(* IEC 61131-3 sources: elnaProjects/ElpcLogic/PomarKc7Changed/build_USO_ecl (part 9) *)

  runDiProtection(protections.dPmaslo_gaz_less100);
  runDiProtection(protections.Reg_vozb_off);
  runDiProtection(protections.Fail_chastotnii_pusk);
  runDiProtection(protections.Off_avar_vikluchatel);
  runDiProtection(protections.AOKC_SHKC);
  runDiProtection(protections.AO_PRU);
  runDiProtection(protections.AO_ot_SHU);
  runDiProtection(protections.mvOff);
  runDiProtection(protections.Kran1_sdvig);
  runDiProtection(protections.Kran2_sdvig);
END_FUNCTION

FUNCTION anyProtectionInRemont : BOOL
  VAR_INPUT
    protections : ProtectionsConfig;
  END_VAR

  anyProtectioninRemont:=
  protections.Topornogo_podshipnika_EDT_1.Remont OR
  protections.Toy_podshipnika_EDT_2.Remont OR
  protections.Toy_podshipnika_kol_EDT_3.remont OR
  protections.Toy_podshipnika_kol_EDT_4.Remont OR
  protections.To_podshipnika_shest_red_EDT_5.Remont OR
  protections.To_podshipnika_shest_red_EDT_6.Remont OR
  protections.To_podshipnika_N_EDT_7.Remont OR
  protections.To_podshipnika_svob_konca_EDT_8.Remont OR
  protections.Ty_podshipnika_rab_kol_EDT_9.Remont OR
  protections.Typornogo_podshipnika_nerab_kolodok_HT_10.Remont OR
  protections.Tgaza_na_vyhode_H.Remont OR
  protections.Os_sdvig_nagnetatelja_plus.Remont OR
  protections.Os_sdvig_nagnetatelja_minus.Remont OR
  protections.Pgaza_na_vyhode_nagnetatelia_GPA_STOP.Remont OR
  protections.Pgaza_na_vhode_nagnetatelia_GPA_STOP.Remont OR
  protections.Pgaza_na_vyhode_nagnetatelia.Remont OR
  protections.dPmaslo_gaz.Remont OR
  protections.Pmaslo_sm_nizkoe.Remont OR
  protections.Pmaslo_sm_vysokoe.Remont OR
  protections.Vibro_skorost_OPED_T1.Remont OR
  protections.Vibro_skorost_OPED_T2.Remont OR
  protections.Vibro_skorost_OYP_kolesa_ED_T3.Remont OR
  protections.Vibro_skorost_OP_kolesa_RH_T4.Remont OR
  protections.Vibro_skorost_OP_shesterni_RED_T5.Remont OR
  protections.Vibro_skorost_OP_shesterni_RED_T6.Remont OR
  protections.dPmaslo_gaz_less100.Remont OR
  protections.Reg_vozb_off.Remont OR
  protections.Fail_chastotnii_pusk.Remont OR
  protections.Off_avar_vikluchatel.Remont OR
  protections.AOKC_SHKC.Remont OR
  protections.AO_PRU.Remont OR
  protections.AO_ot_SHU.Remont OR
  protections.mvOff.Remont OR
  protections.Kran1_sdvig.Remont OR
  protections.Kran2_sdvig.Remont;
END_FUNCTION

FUNCTION ResetAllSignaling : BOOL
  VAR_IN_OUT
    protections : ProtectionsConfig;
  END_VAR

  IF protections.Topornogo_podshipnika_EDT_1.Signaling THEN
      resetAiProtection(protections.Topornogo_podshipnika_EDT_1);  END_IF;

  IF protections.Toy_podshipnika_EDT_2.Signaling THEN
      resetAiProtection(protections.Toy_podshipnika_EDT_2); END_IF;

  IF protections.Toy_podshipnika_kol_EDT_3.Signaling THEN
      resetAiProtection(protections.Toy_podshipnika_kol_EDT_3); END_IF;

  IF protections.Toy_podshipnika_kol_EDT_4.Signaling THEN
      resetAiProtection(protections.Toy_podshipnika_kol_EDT_4); END_IF;

  IF protections.To_podshipnika_shest_red_EDT_5.Signaling THEN
      resetAiProtection(protections.To_podshipnika_shest_red_EDT_5); END_IF;

  IF protections.To_podshipnika_shest_red_EDT_6.Signaling THEN
      resetAiProtection(protections.To_podshipnika_shest_red_EDT_6); END_IF;

  IF protections.To_podshipnika_N_EDT_7.Signaling THEN
      resetAiProtection(protections.To_podshipnika_N_EDT_7); END_IF;

  IF protections.To_podshipnika_svob_konca_EDT_8.Signaling THEN
      resetAiProtection(protections.To_podshipnika_svob_konca_EDT_8); END_IF;

  IF protections.Ty_podshipnika_rab_kol_EDT_9.Signaling THEN
      resetAiProtection(protections.Ty_podshipnika_rab_kol_EDT_9); END_IF;

  IF protections.Typornogo_podshipnika_nerab_kolodok_HT_10.Signaling THEN
      resetAiProtection(protections.Typornogo_podshipnika_nerab_kolodok_HT_10); END_IF;

  IF protections.Tgaza_na_vyhode_H.Signaling THEN
      resetAiProtection(protections.Tgaza_na_vyhode_H); END_IF;

  IF protections.Os_sdvig_nagnetatelja_plus.Signaling THEN
     resetAiProtection(protections.Os_sdvig_nagnetatelja_plus); END_IF;

  IF protections.Os_sdvig_nagnetatelja_minus.Signaling THEN
      resetAiProtection(protections.Os_sdvig_nagnetatelja_minus); END_IF;

  IF protections.Pgaza_na_vyhode_nagnetatelia_GPA_STOP.Signaling THEN
      resetAiProtection(protections.Pgaza_na_vyhode_nagnetatelia_GPA_STOP); END_IF;

  IF protections.Pgaza_na_vhode_nagnetatelia_GPA_STOP.Signaling THEN
      resetAiProtection(protections.Pgaza_na_vhode_nagnetatelia_GPA_STOP); END_IF;

  IF protections.Pgaza_na_vyhode_nagnetatelia.Signaling THEN
      resetAiProtection(protections.Pgaza_na_vyhode_nagnetatelia); END_IF;

  IF protections.dPmaslo_gaz.Signaling THEN
      resetAiProtection(protections.dPmaslo_gaz); END_IF;

  IF protections.Pmaslo_sm_nizkoe.Signaling THEN
      resetAiProtection(protections.Pmaslo_sm_nizkoe); END_IF;

  IF protections.Pmaslo_sm_vysokoe.Signaling THEN
      resetAiProtection(protections.Pmaslo_sm_vysokoe); END_IF;

  IF protections.Vibro_skorost_OPED_T1.Signaling THEN
      resetAiProtection(protections.Vibro_skorost_OPED_T1); END_IF;

  IF protections.Vibro_skorost_OPED_T2.Signaling THEN
      resetAiProtection(protections.Vibro_skorost_OPED_T2); END_IF;

  IF protections.Vibro_skorost_OYP_kolesa_ED_T3.Signaling THEN
      resetAiProtection(protections.Vibro_skorost_OYP_kolesa_ED_T3); END_IF;

  IF protections.Vibro_skorost_OP_kolesa_RH_T4.Signaling THEN
      resetAiProtection(protections.Vibro_skorost_OP_kolesa_RH_T4); END_IF;

  IF protections.Vibro_skorost_OP_shesterni_RED_T5.Signaling THEN
      resetAiProtection(protections.Vibro_skorost_OP_shesterni_RED_T5); END_IF;

  IF protections.Vibro_skorost_OP_shesterni_RED_T6.Signaling THEN
      resetAiProtection(protections.Vibro_skorost_OP_shesterni_RED_T6); END_IF;

  IF protections.dPmaslo_gaz_less100.Signaling THEN
      resetDiProtection(protections.dPmaslo_gaz_less100); END_IF;

  IF protections.Reg_vozb_off.Signaling THEN
      resetDiProtection(protections.Reg_vozb_off); END_IF;

  IF protections.Fail_chastotnii_pusk.Signaling THEN
      resetDiProtection(protections.Fail_chastotnii_pusk); END_IF;

  IF protections.Off_avar_vikluchatel.Signaling THEN
      resetDiProtection(protections.Off_avar_vikluchatel); END_IF;

  IF protections.AOKC_SHKC.Signaling THEN
      resetDiProtection(protections.AOKC_SHKC); END_IF;

  IF protections.AO_PRU.Signaling THEN
      resetDiProtection(protections.AO_PRU); END_IF;

  IF protections.AO_ot_SHU.Signaling THEN
      resetDiProtection(protections.AO_ot_SHU); END_IF;

  IF protections.mvOff.Signaling THEN
      resetDiProtection(protections.mvOff); END_IF;

  IF protections.Kran1_sdvig.Signaling THEN
      resetDiProtection(protections.Kran1_sdvig); END_IF;

  IF protections.Kran2_sdvig.Signaling THEN
      resetDiProtection(protections.Kran2_sdvig); END_IF;
END_FUNCTION

FUNCTION_BLOCK fb_ProtectionsManager
  VAR
    cmd : BYTE;
  END_VAR
  VAR_IN_OUT
    str_PM : struct_ProtectionsManager;
  END_VAR
  VAR
    lastCmd : BYTE;
    autoRunPriznak : BOOL;
    onInit : BOOL;
  END_VAR
  VAR_EXTERNAL
    protections : ProtectionsConfig;
  END_VAR
  VAR
    timerUnBlock : TON;
    timerAutoRun : TON;
    UnBlockPriznak : BOOL;
  END_VAR

  IF NOT onInit THEN

      autoRunProtections(protections);
  onInit:=TRUE;
  END_IF;

  str_PM.protectionInRemont:=anyProtectioninRemont(protections);

  cmd := str_PM.inCommand;

  IF cmd <> 0 AND lastCmd <> cmd then
                UnBlockPriznak:=TRUE;
  	CASE BYTE_TO_INT(cmd) OF

  		(*RestartAllSignaling*) 1: 	ResetAllSignaling(protections);
  				          autoRunPriznak:=TRUE;

  	        (*RestartAllProtections*) 2: 	ResetAllProtections(protections);
                                                    autoRunPriznak:=TRUE;

                        (*CheckProtections*)  3: 	RunAllProtections(protections);

  	         (*ResetAllProtections*)  4: 	ResetAllProtections(protections);

  	END_CASE;

  END_IF;
  lastCmd := cmd;
  timerUnBlock(IN:=UnBlockPriznak, PT:=T#1S);
  timerAutoRun(IN:=autoRunPriznak, PT:=T#500MS);

  IF timerAutoRun.Q THEN autoRunProtections(protections);
  END_IF;

  IF timerUnBlock.Q THEN
  lastCmd:= 0;
  str_PM.inCommand:=0;
  autoRunPriznak:=FALSE;
  UnBlockPriznak:=FALSE;
  END_IF;
END_FUNCTION_BLOCK

FUNCTION stopPusk : BOOL
  VAR_IN_OUT
    algoritms : AlgoritmsConfig;
  END_VAR

  resetAndDisable(alg:=algoritms.Apusk);
  resetAndDisable(alg:=algoritms.SemiAutoPusk);
  resetAndDisable(alg:=algoritms.testPms);
  resetAndDisable(alg:=algoritms.puskV);
  resetAndDisable(alg:=algoritms.puskK);
  resetAndDisable(alg:=algoritms.testdPmg);
  resetAndDisable(alg:=algoritms.ppu);
  resetAndDisable(alg:=algoritms.puskOilSystem);
  resetAndDisable(alg:=algoritms.filling);
  resetAndDisable(alg:=algoritms.engineRun);
  resetAndDisable(alg:=algoritms.RingToLine);
  resetAndDisable(alg:=algoritms.LineToRing);
END_FUNCTION

FUNCTION anyDiscretPS : BOOL
  VAR_INPUT
    im : ImConfig;
  END_VAR

  anyDiscretPS:= TRUE;
      (*Im.SingleSignals.BEAO_srabotal.Q                     OR
      Im.SingleSignals.Vozb_ProboiVentila.Q	 OR
      Im.SingleSignals.Vozb_AsinchHod.Q	           OR
      Im.SingleSignals.NS_ForsingVozbugdenia.Q       OR
      Im.SingleSignals.Vozb_AutoUprVozbuditela_off.Q OR
      Im.SingleSignals.Vozb_KontaktorON.Q*)
END_FUNCTION

FUNCTION UnBlockAllProtections : BOOL
  VAR_IN_OUT
    protections : ProtectionsConfig;
  END_VAR

  protections.Topornogo_podshipnika_EDT_1.inOpcCommandsDisabled:=FALSE;
  protections.Toy_podshipnika_EDT_2.inOpcCommandsDisabled:=FALSE;
  protections.Toy_podshipnika_kol_EDT_3.inOpcCommandsDisabled:=FALSE;
  protections.Toy_podshipnika_kol_EDT_4.inOpcCommandsDisabled:=FALSE;
  protections.To_podshipnika_shest_red_EDT_5.inOpcCommandsDisabled:=FALSE;
  protections.To_podshipnika_shest_red_EDT_6.inOpcCommandsDisabled:=FALSE;
  protections.To_podshipnika_N_EDT_7.inOpcCommandsDisabled:=FALSE;
  protections.To_podshipnika_svob_konca_EDT_8.inOpcCommandsDisabled:=FALSE;
  protections.Ty_podshipnika_rab_kol_EDT_9.inOpcCommandsDisabled:=FALSE;
  protections.Typornogo_podshipnika_nerab_kolodok_HT_10.inOpcCommandsDisabled:=FALSE;
  protections.Tgaza_na_vyhode_H.inOpcCommandsDisabled:=FALSE;
  protections.Os_sdvig_nagnetatelja_plus.inOpcCommandsDisabled:=FALSE;
  protections.Os_sdvig_nagnetatelja_minus.inOpcCommandsDisabled:=FALSE;
  protections.Pgaza_na_vyhode_nagnetatelia_GPA_STOP.inOpcCommandsDisabled:=FALSE;
  protections.Pgaza_na_vhode_nagnetatelia_GPA_STOP.inOpcCommandsDisabled:=FALSE;
  protections.Pgaza_na_vyhode_nagnetatelia.inOpcCommandsDisabled:=FALSE;
  protections.dPmaslo_gaz.inOpcCommandsDisabled:=FALSE;
  protections.Pmaslo_sm_nizkoe.inOpcCommandsDisabled:=FALSE;
  protections.Pmaslo_sm_vysokoe.inOpcCommandsDisabled:=FALSE;
  protections.Vibro_skorost_OPED_T1.inOpcCommandsDisabled:=FALSE;
  protections.Vibro_skorost_OPED_T2.inOpcCommandsDisabled:=FALSE;
  protections.Vibro_skorost_OYP_kolesa_ED_T3.inOpcCommandsDisabled:=FALSE;
  protections.Vibro_skorost_OP_kolesa_RH_T4.inOpcCommandsDisabled:=FALSE;
  protections.Vibro_skorost_OP_shesterni_RED_T5.inOpcCommandsDisabled:=FALSE;
  protections.Vibro_skorost_OP_shesterni_RED_T6.inOpcCommandsDisabled:=FALSE;
  protections.dPmaslo_gaz_less100.inOpcCommandsDisabled:=FALSE;
  protections.Reg_vozb_off.inOpcCommandsDisabled:=FALSE;
  protections.Fail_chastotnii_pusk.inOpcCommandsDisabled:=FALSE;
  protections.Off_avar_vikluchatel.inOpcCommandsDisabled:=FALSE;
  protections.AOKC_SHKC.inOpcCommandsDisabled:=FALSE;
  protections.AO_PRU.inOpcCommandsDisabled:=FALSE;
  protections.AO_ot_SHU.inOpcCommandsDisabled:=FALSE;
  protections.mvOff.inOpcCommandsDisabled:=FALSE;
  protections.Kran1_sdvig.inOpcCommandsDisabled:=FALSE;
  protections.Kran2_sdvig.inOpcCommandsDisabled:=FALSE;
END_FUNCTION

FUNCTION_BLOCK fb_AlgoritmsManager
  VAR_IN_OUT
    str_AM : struct_AlgoritmsManager;
  END_VAR
  VAR
    onInit : BOOL;
  END_VAR
  VAR_EXTERNAL
    ai : AiConfig;
  END_VAR
  VAR
    EoTrig : R_TRIG;
    EoFTrig : F_TRIG;
    PsLampTrig : R_TRIG;
    PsLampFTrig : F_TRIG;
    Ring : R_TRIG;
    Line : R_TRIG;
    statusDualInput : TYPE_statusDualInput;
  END_VAR
  VAR_EXTERNAL
    IM : ImConfig;
    protections : ProtectionsConfig;
    algoritms : AlgoritmsConfig;
    ModeGpa : TYPE_ModeGpa;
  END_VAR

  IF NOT onInit THEN
            DisableAiLimits(ai);
            (*IM.SingleSignals.P_oil_low.Disabled_Sig:=TRUE;
            IM.SingleSignals.dP_oilgaz_low.Disabled_Sig:=TRUE;*)
            str_AM.nMode:=ModeGpa.MODE_STOP;
            BlockAllIM(IM);
            runIfNotRunning(algoritms.AutoTen);
  onInit:=TRUE;
  END_IF;

  str_AM.DiscretPS:=anyDiscretPS(IM);
  str_AM.AnalogsPs:=anyAnalogsPs(ai);
  str_AM.ProtectionSignaling:=anyProtectionSignaling(protections);

  (*EoTrig(CLK := IM.SingleSignals.BEO_Srabat.Q);*)
  IF EoTrig.Q THEN
  	stopPusk(algoritms);
  	resetAndDisable(algoritms.Remont);
  	resetAndDisable(algoritms.no);
  	resetAndDisable(algoritms.ao);
  	str_AM.nMode:=ModeGpa.MODE_EO;
  END_IF;
  (*EoFTrig(CLK := IM.SingleSignals.BEO_Srabat.Q);*)
  IF EoFTrig.Q THEN
  	str_AM.nMode:=ModeGpa.MODE_STOP;
  	runIfNotRunning(algoritms.ao);
  END_IF;

  (*IF (str_AM.ProtectionSignaling OR Im.SingleSignals.AO_KC.Q OR Im.SingleSignals.AOGPA_knopkaSHU.Q OR Im.SingleSignals.AOGPA_PRU.Q )
  	AND NOT((str_AM.mode=ModeGpa.MODE_AO) OR (str_AM.mode=ModeGpa.MODE_EO) OR IM.SingleOutputs.IndikicijaAS_fonar.Q
            OR (str_AM.mode=ModeGpa.MODE_TESTAZ) OR (str_AM.mode=ModeGpa.MODE_TESTDPMG) OR (str_AM.mode=ModeGpa.MODE_REMONT) OR
            (str_AM.mode=ModeGpa.MODE_TESTPMS))THEN
  		runIfNotRunning(algoritms.ao);
  	str_AM.nMode:=ModeGpa.MODE_AO;
  END_IF;
  *)
  (*IF Im.SingleSignals.NOGPA_knopkaSHU.Q  AND algoritms.no.CanRun THEN
  	runIfNotRunning(algoritms.no);
            str_AM.nMode:=ModeGpa.MODE_NO;
  END_IF;*)

  PsLampTrig(CLK := str_AM.DiscretPS OR str_AM.AnalogsPs);
  (*IF PsLampTrig.Q THEN
            runIfNotRunningSO(IM.SingleOutputs.IndikicijaPS_fonar);
  END_IF;*)
  PsLampFTrig(CLK := str_AM.DiscretPS OR str_AM.AnalogsPs);
  (*IF PsLampFTrig.Q THEN
            resetIfRunningSO(IM.SingleOutputs.IndikicijaPS_fonar);
  END_IF;*)

  IF str_AM.mode = ModeGpa.MODE_WORK_Line OR str_AM.mode = ModeGpa.MODE_WORK_Ring  THEN

  	Ring(CLK:=Im.kran6.onStatus=statusDualInput.STATUS_On);
  	Line(CLK:=Im.kran6.onStatus=statusDualInput.STATUS_Off);

  	IF Ring.Q AND str_AM.mode = ModeGpa.MODE_WORK_Line THEN
  		str_AM.nMode:=ModeGpa.MODE_WORK_Ring;
  	END_IF;
  	IF Line.Q AND str_AM.mode = ModeGpa.MODE_WORK_Ring THEN
  		str_AM.nMode:=ModeGpa.MODE_WORK_Line;
  	END_IF;

  END_IF;

  IF str_AM.mode = ModeGpa.MODE_WORK_Line THEN
            runIfNotRunning(alg:=algoritms.AntiPompag);
  	ELSE
            resetAndDisable(alg:=algoritms.AntiPompag);
  END_IF;

  IF str_AM.nMode<>str_AM.mode THEN
  	str_AM.mode:=str_AM.nMode;
  	CASE str_AM.mode OF
  	(*ModeGpa.MODE_REMONT*)1:
  		stopPusk(algoritms);
  		resetAndDisable(alg:=algoritms.no);
  		resetAndDisable(alg:=algoritms.ao);
  		resetAndDisable(alg:=algoritms.TestProtection);
                      resetAndDisable(alg:=algoritms.testIm);

  	(*ModeGpa.MODE_TESTAZ*)16:
  		stopPusk(algoritms);
  		resetAndDisable(alg:=algoritms.ao);
  		resetAndDisable(alg:=algoritms.no);
                      resetAndDisable(alg:=algoritms.Remont);
                      resetAndDisable(alg:=algoritms.testIm);

            (*ModeGpa.MODE_TESTIM*)15:
                      stopPusk(algoritms);
                      resetAndDisable(alg:=algoritms.Remont);
                      resetAndDisable(alg:=algoritms.TestProtection);

  	(*ModeGpa.MODE_EO*)14:
  		stopPusk(algoritms);
  		resetAndDisable(alg:=algoritms.no);
  		resetAndDisable(alg:=algoritms.ao);
  		resetAndDisable(alg:=algoritms.Remont);
                      resetAndDisable(alg:=algoritms.testIm);
                      resetAndDisable(alg:=algoritms.TestProtection);
  	(*ModeGpa.MODE_AO*)13:
  		(*//stopPusk();*)
  		resetAndDisable(alg:=algoritms.no);
  		resetAndDisable(alg:=algoritms.Remont);
                      resetAndDisable(alg:=algoritms.testIm);
                      resetAndDisable(alg:=algoritms.TestProtection);
                      algoritms.VibegPNS.inCanRun:=TRUE;
  	(*ModeGpa.MODE_NO*)12:
  		stopPusk(algoritms);
                      resetAndDisable(alg:=algoritms.testIm);
                      resetAndDisable(alg:=algoritms.Remont);
                      resetAndDisable(alg:=algoritms.TestProtection);
                      algoritms.VibegPNS.inCanRun:=TRUE;
  		algoritms.ao.inCanRun:=TRUE;
  	(*ModeGpa.MODE_APUSK*)8:
  		resetAndDisable(alg:=algoritms.SemiAutoPusk);
  		resetAndDisable(alg:=algoritms.puskV);
  		resetAndDisable(alg:=algoritms.puskK);
  		resetAndDisable(alg:=algoritms.testdPmg);
  		resetAndDisable(alg:=algoritms.testPms);
  		(*resetAndDisable(alg:=algoritms.testIm);
                      resetAndDisable(alg:=algoritms.TestProtection);
                      resetAndDisable(alg:=algoritms.Remont);*)
  		resetAndDisable(alg:=algoritms.ppu);
  		algoritms.no.inCanRun:=TRUE;
  		algoritms.ao.inCanRun:=TRUE;

  	(*ModeGpa.MODE_MPUSK*)9:
  		resetAndDisable(alg:=algoritms.Apusk);
  		resetAndDisable(alg:=algoritms.puskV);
  		resetAndDisable(alg:=algoritms.puskK);
  		resetAndDisable(alg:=algoritms.testdPmg);
  		resetAndDisable(alg:=algoritms.testPms);
  		(*resetAndDisable(alg:=algoritms.testIm);
                      resetAndDisable(alg:=algoritms.TestProtection);
                      resetAndDisable(alg:=algoritms.Remont);	*)
  		resetAndDisable(alg:=algoritms.ppu);
  		algoritms.no.inCanRun:=TRUE;
                      algoritms.no.inOpcCommandsDisabled:=FALSE;
  		algoritms.ao.inCanRun:=TRUE;
                      algoritms.ao.inOpcCommandsDisabled:=FALSE;

  	(*ModeGpa.MODE_PUSKK*)5:
                      resetAndDisable(alg:=algoritms.ppu);
  		resetAndDisable(alg:=algoritms.Apusk);
  		resetAndDisable(alg:=algoritms.SemiAutoPusk);
  		resetAndDisable(alg:=algoritms.TestProtection);
                      resetAndDisable(alg:=algoritms.Remont);
  		resetAndDisable(alg:=algoritms.testIm	 );
  		algoritms.no.inCanRun:=TRUE;
                      algoritms.no.inOpcCommandsDisabled:=FALSE;
  		algoritms.ao.inCanRun:=TRUE;
                      algoritms.ao.inOpcCommandsDisabled:=FALSE;
  	(*ModeGpa.MODE_PUSKV*)4:
                      resetAndDisable(alg:=algoritms.ppu);
  		resetAndDisable(alg:=algoritms.Apusk);
  		resetAndDisable(alg:=algoritms.SemiAutoPusk);
  		resetAndDisable(alg:=algoritms.TestProtection);
                      resetAndDisable(alg:=algoritms.Remont);
  		resetAndDisable(alg:=algoritms.testIm	 );
  		algoritms.no.inCanRun:=TRUE;
                      algoritms.no.inOpcCommandsDisabled:=FALSE;
  		algoritms.ao.inCanRun:=TRUE;
                      algoritms.ao.inOpcCommandsDisabled:=FALSE;

  	(*ModeGpa.MODE_TESTDPMG*)6:
                      resetAndDisable(alg:=algoritms.ppu);
  		resetAndDisable(alg:=algoritms.Apusk);
  		resetAndDisable(alg:=algoritms.SemiAutoPusk);
  		resetAndDisable(alg:=algoritms.TestProtection);
                      resetAndDisable(alg:=algoritms.Remont);
  		resetAndDisable(alg:=algoritms.testIm	 );
  		algoritms.no.inCanRun:=TRUE;
                      algoritms.no.inOpcCommandsDisabled:=FALSE;
  		algoritms.ao.inCanRun:=TRUE;
                      algoritms.ao.inOpcCommandsDisabled:=FALSE;

  	(*ModeGpa.MODE_TESTPMS*)7:
                      resetAndDisable(alg:=algoritms.ppu);
  		resetAndDisable(alg:=algoritms.Apusk);
  		resetAndDisable(alg:=algoritms.SemiAutoPusk);
  		resetAndDisable(alg:=algoritms.TestProtection);
                      resetAndDisable(alg:=algoritms.Remont);
  		resetAndDisable(alg:=algoritms.testIm);
  		algoritms.no.inCanRun:=TRUE;
                      algoritms.no.inOpcCommandsDisabled:=FALSE;
  		algoritms.ao.inCanRun:=TRUE;
                      algoritms.ao.inOpcCommandsDisabled:=FALSE;

  	(*ModeGpa.MODE_WORK_Ring*)10:
  		resetAndDisable(alg:=algoritms.Apusk);
  		resetAndDisable(alg:=algoritms.SemiAutoPusk);
  		resetAndDisable(alg:=algoritms.puskV);
  		resetAndDisable(alg:=algoritms.puskK);
  		resetAndDisable(alg:=algoritms.testdPmg);
  		resetAndDisable(alg:=algoritms.testPms);
  		resetAndDisable(alg:=algoritms.ppu);
  		algoritms.no.inCanRun:=TRUE;
                      algoritms.no.inOpcCommandsDisabled:=FALSE;
  		algoritms.ao.inCanRun:=TRUE;
                      algoritms.ao.inOpcCommandsDisabled:=FALSE;

  	(*ModeGpa.MODE_WORK_Line*)11:
  		resetAndDisable(alg:=algoritms.Apusk);
  		resetAndDisable(alg:=algoritms.SemiAutoPusk);
  		resetAndDisable(alg:=algoritms.puskV);
  		resetAndDisable(alg:=algoritms.puskK);
  		resetAndDisable(alg:=algoritms.testdPmg);
  		resetAndDisable(alg:=algoritms.testPms);
  		resetAndDisable(alg:=algoritms.ppu);
  		resetAndDisable(alg:=algoritms.testIm	 );
  		algoritms.no.inCanRun:=TRUE;
                      algoritms.no.inOpcCommandsDisabled:=FALSE;
  		algoritms.ao.inCanRun:=TRUE;
                      algoritms.ao.inOpcCommandsDisabled:=FALSE;

  	(*ModeGpa.MODE_STOP*)2:
  		algoritms.ppu.inCanRun:=TRUE;
                      runIfNotRunning(alg:=algoritms.ppu);
  		algoritms.no.inCanRun:=TRUE;
                      algoritms.no.inOpcCommandsDisabled:=FALSE;
  		algoritms.ao.inCanRun:=TRUE;
                      algoritms.ao.inOpcCommandsDisabled:=FALSE;
                      (*UnBlockAllProtections(protections);*)
  		BlockAllIM(IM);
  		algoritms.Remont.inCanRun:=TRUE;
  		algoritms.Remont.inOpcCommandsDisabled:=FALSE;
  		algoritms.testim.inCanRun:=TRUE;
  		algoritms.testim.inOpcCommandsDisabled:=FALSE;
  		algoritms.TestProtection.inCanRun:=TRUE;
  		algoritms.TestProtection.inOpcCommandsDisabled:=FALSE;
                      algoritms.VibegPNS.inCanRun:=FALSE;
                      algoritms.AutoAvom.inCanRun:=FALSE;
  		(*resetAndDisable(alg:=algoritms.puskV);
  		resetAndDisable(alg:=algoritms.puskK);
  		resetAndDisable(alg:=algoritms.testdPmg);
  		resetAndDisable(alg:=algoritms.testPms);*)
  	(*ModeGpa.MODE_READY*)3:
  		resetAndDisable(alg:=algoritms.Remont);
  		resetAndDisable(alg:=algoritms.testim);
  		resetAndDisable(alg:=algoritms.TestProtection);
                      algoritms.Apusk.inCanRun:=TRUE;
                      algoritms.Apusk.inOpcCommandsDisabled:=FALSE;
  		algoritms.SemiAutoPusk.inCanRun:=TRUE;
                      algoritms.SemiAutoPusk.inOpcCommandsDisabled:=FALSE;
  	END_CASE;
  END_IF;
END_FUNCTION_BLOCK

FUNCTION remontAllProtections : BOOL
  VAR_IN_OUT
    protections : ProtectionsConfig;
  END_VAR
  VAR CONSTANT
    cmdRemont : WORD          := 4;
  END_VAR

  protections.Topornogo_podshipnika_EDT_1.inCommand_Alg:=cmdRemont;
  protections.Toy_podshipnika_EDT_2.inCommand_Alg:=cmdRemont;
  protections.Toy_podshipnika_kol_EDT_3.inCommand_Alg:=cmdRemont;
  protections.Toy_podshipnika_kol_EDT_4.inCommand_Alg:=cmdRemont;
  protections.To_podshipnika_shest_red_EDT_5.inCommand_Alg:=cmdRemont;
  protections.To_podshipnika_shest_red_EDT_6.inCommand_Alg:=cmdRemont;
  protections.To_podshipnika_N_EDT_7.inCommand_Alg:=cmdRemont;
  protections.To_podshipnika_svob_konca_EDT_8.inCommand_Alg:=cmdRemont;
  protections.Ty_podshipnika_rab_kol_EDT_9.inCommand_Alg:=cmdRemont;
  protections.Typornogo_podshipnika_nerab_kolodok_HT_10.inCommand_Alg:=cmdRemont;
  protections.Tgaza_na_vyhode_H.inCommand_Alg:=cmdRemont;
  protections.Os_sdvig_nagnetatelja_plus.inCommand_Alg:=cmdRemont;
  protections.Os_sdvig_nagnetatelja_minus.inCommand_Alg:=cmdRemont;
  protections.Pgaza_na_vyhode_nagnetatelia_GPA_STOP.inCommand_Alg:=cmdRemont;
  protections.Pgaza_na_vhode_nagnetatelia_GPA_STOP.inCommand_Alg:=cmdRemont;
  protections.Pgaza_na_vyhode_nagnetatelia.inCommand_Alg:=cmdRemont;
  protections.dPmaslo_gaz.inCommand_Alg:=cmdRemont;
  protections.Pmaslo_sm_nizkoe.inCommand_Alg:=cmdRemont;
  protections.Pmaslo_sm_vysokoe.inCommand_Alg:=cmdRemont;
  protections.Vibro_skorost_OPED_T1.inCommand_Alg:=cmdRemont;
  protections.Vibro_skorost_OPED_T2.inCommand_Alg:=cmdRemont;
  protections.Vibro_skorost_OYP_kolesa_ED_T3.inCommand_Alg:=cmdRemont;
  protections.Vibro_skorost_OP_kolesa_RH_T4.inCommand_Alg:=cmdRemont;
  protections.Vibro_skorost_OP_shesterni_RED_T5.inCommand_Alg:=cmdRemont;
  protections.Vibro_skorost_OP_shesterni_RED_T6.inCommand_Alg:=cmdRemont;
  protections.dPmaslo_gaz_less100.inCommand_Alg:=cmdRemont;
  protections.Reg_vozb_off.inCommand_Alg:=cmdRemont;
  protections.Fail_chastotnii_pusk.inCommand_Alg:=cmdRemont;
  protections.Off_avar_vikluchatel.inCommand_Alg:=cmdRemont;
  protections.AOKC_SHKC.inCommand_Alg:=cmdRemont;
  protections.AO_PRU.inCommand_Alg:=cmdRemont;
  protections.AO_ot_SHU.inCommand_Alg:=cmdRemont;
  protections.mvOff.inCommand_Alg:=cmdRemont;
  protections.Kran1_sdvig.inCommand_Alg:=cmdRemont;
  protections.Kran2_sdvig.inCommand_Alg:=cmdRemont;
END_FUNCTION

FUNCTION nsCepeiControl : BOOL
  VAR_INPUT
    im : ImConfig;
  END_VAR

  nsCepeiControl:= NOT (
  	im.kran1.reliability OR
  	im.kran2.reliability OR
  	im.kran4.reliability OR
  	im.kran5.reliability OR
  	im.kran6.reliability OR
  	im.kran3b.reliability OR
  	im.pns.reliability OR
  	im.nu1.reliability OR
  	im.nu2.reliability OR
  	im.PNS.reliability OR
            im.v1_Avom.reliability OR
            im.v2_Avom.reliability OR
            (*im.Ten.reliability OR*)
  	im.mv.reliability);
END_FUNCTION

FUNCTION NapryageniaOK : BOOL
  VAR_INPUT
    im : ImConfig;
  END_VAR

  NapryageniaOK:=
  NOT (Im.SingleSignals.NS_G1_G2.Q
  OR Im.SingleSignals.NS_G10_G11.Q
  OR Im.SingleSignals.NS_G13_G14.Q
  OR Im.SingleSignals.NS_G15_G16.Q
  OR Im.SingleSignals.NS_G17.Q
  OR Im.SingleSignals.NS_G18_G19.Q
  OR Im.SingleSignals.NS_G3_G4.Q
  OR Im.SingleSignals.NS_G5_G6.Q
  OR Im.SingleSignals.NS_G7_G8.Q
  OR im.SingleSignals.QF1_on.Q
  OR Im.SingleSignals.QF2_on.Q
  OR Im.SingleSignals.QF23_on.Q
  OR Im.SingleSignals.QF4_QF5_on.Q
  OR Im.SingleSignals.QF6_QF7_on.Q
  OR Im.SingleSignals.QF8_QF9_on.Q
  OR Im.SingleSignals.QF10_QF11_on.Q
  OR im.SingleSignals.QF12_QF13_on.Q
  OR im.SingleSignals.QF22_on.Q
  OR Im.SingleSignals.QF14_QF15_on.Q);
END_FUNCTION

FUNCTION discretNS : BOOL
  VAR_INPUT
    di : DiConfig;
  END_VAR

  discretNS:=  ((di.di_0.reliability <> 255)
                OR (di.di_1.reliability <> 255)
                OR (di.di_2.reliability <> 255)
                OR (di.di_3.reliability <> 255)
                OR (di.di_4.reliability <> 255)
                OR (di.di_5.reliability <> 255)
                OR (di.di_6.reliability <> 255)
                OR (di.di_7.reliability <> 255)
                OR (di.di_8.reliability <> 255)
                OR (di.di_9.reliability <> 255)
                OR (di.di_10.reliability <> 255)
                OR (di.di_11.reliability <> 255)
                OR (di.di_12.reliability <> 255)
                OR (di.di_13.reliability <> 255)
                OR (di.di_14.reliability <> 255));
               (* OR (di.di_15.reliability <> 255)); *)
END_FUNCTION

FUNCTION BlockAllProtections : BOOL
  VAR_IN_OUT
    protections : ProtectionsConfig;
  END_VAR

  protections.Topornogo_podshipnika_EDT_1.inOpcCommandsDisabled:=TRUE;
  protections.Toy_podshipnika_EDT_2.inOpcCommandsDisabled:=TRUE;
  protections.Toy_podshipnika_kol_EDT_3.inOpcCommandsDisabled:=TRUE;
  protections.Toy_podshipnika_kol_EDT_4.inOpcCommandsDisabled:=TRUE;
  protections.To_podshipnika_shest_red_EDT_5.inOpcCommandsDisabled:=TRUE;
  protections.To_podshipnika_shest_red_EDT_6.inOpcCommandsDisabled:=TRUE;
  protections.To_podshipnika_N_EDT_7.inOpcCommandsDisabled:=TRUE;
  protections.To_podshipnika_svob_konca_EDT_8.inOpcCommandsDisabled:=TRUE;
  protections.Ty_podshipnika_rab_kol_EDT_9.inOpcCommandsDisabled:=TRUE;
  protections.Typornogo_podshipnika_nerab_kolodok_HT_10.inOpcCommandsDisabled:=TRUE;
  protections.Tgaza_na_vyhode_H.inOpcCommandsDisabled:=TRUE;
  protections.Os_sdvig_nagnetatelja_plus.inOpcCommandsDisabled:=TRUE;
  protections.Os_sdvig_nagnetatelja_minus.inOpcCommandsDisabled:=TRUE;
  protections.Pgaza_na_vyhode_nagnetatelia_GPA_STOP.inOpcCommandsDisabled:=TRUE;
  protections.Pgaza_na_vhode_nagnetatelia_GPA_STOP.inOpcCommandsDisabled:=TRUE;
  protections.Pgaza_na_vyhode_nagnetatelia.inOpcCommandsDisabled:=TRUE;
  protections.dPmaslo_gaz.inOpcCommandsDisabled:=TRUE;
  protections.Pmaslo_sm_nizkoe.inOpcCommandsDisabled:=TRUE;
  protections.Pmaslo_sm_vysokoe.inOpcCommandsDisabled:=TRUE;
  protections.Vibro_skorost_OPED_T1.inOpcCommandsDisabled:=TRUE;
  protections.Vibro_skorost_OPED_T2.inOpcCommandsDisabled:=TRUE;
  protections.Vibro_skorost_OYP_kolesa_ED_T3.inOpcCommandsDisabled:=TRUE;
  protections.Vibro_skorost_OP_kolesa_RH_T4.inOpcCommandsDisabled:=TRUE;
  protections.Vibro_skorost_OP_shesterni_RED_T5.inOpcCommandsDisabled:=TRUE;
  protections.Vibro_skorost_OP_shesterni_RED_T6.inOpcCommandsDisabled:=TRUE;
  protections.dPmaslo_gaz_less100.inOpcCommandsDisabled:=TRUE;
  protections.Reg_vozb_off.inOpcCommandsDisabled:=TRUE;
  protections.Fail_chastotnii_pusk.inOpcCommandsDisabled:=TRUE;
  protections.Off_avar_vikluchatel.inOpcCommandsDisabled:=TRUE;
  protections.AOKC_SHKC.inOpcCommandsDisabled:=TRUE;
  protections.AO_PRU.inOpcCommandsDisabled:=TRUE;
  protections.AO_ot_SHU.inOpcCommandsDisabled:=TRUE;
  protections.mvOff.inOpcCommandsDisabled:=TRUE;
  protections.Kran1_sdvig.inOpcCommandsDisabled:=TRUE;
  protections.Kran2_sdvig.inOpcCommandsDisabled:=TRUE;
END_FUNCTION

PROGRAM program0
  VAR
    SysTime : LREAL;
    systime_ns : ULINT;
    systime_s : ULINT;
    preSysTime : LREAL;
    tmpCycle : LREAL;
    preSys_s : ULINT;
    preSys_ns : ULINT;
  END_VAR
  VAR_EXTERNAL
    cur_Cycle : REAL;
    gStart_Tmr : REAL;
  END_VAR
  VAR
    Timings : fb_Timings;
    _init : BOOL          := TRUE;
    life_count : UINT;
    AI_structs_ini : proc_AI_Init;
    AI_Proc : proc_AI;
    AO_structs_ini : proc_AO_Init;
    AO_Proc : proc_AO;
    DI_structs_ini : proc_DI_Init;
    DI_Proc : proc_DI;
    DO_structs_ini : proc_DO_Init;
    DO_Proc : proc_DO;
    Get_algoritms_OPC : OPC_algoritms_set;
    Set_algoritms_OPC : OPC_algoritms_get;
    IM_structs_ini : proc_IM_Init;
    IM_Proc : proc_IM;
    Protections_structs_ini : proc_Protections_Init;
    Protections_Proc : proc_Protection;
    Algoritms_Proc : proc_algoritms;
    AlgoritmsManager : fb_AlgoritmsManager;
    ProtectionsManager : fb_ProtectionsManager;
  END_VAR
  VAR_EXTERNAL
    algManager : struct_AlgoritmsManager;
    protectManager : struct_ProtectionsManager;
  END_VAR

  (* Обработка времени. *)
  SysTime := ULINT_TO_LREAL(systime_s) + (1.0E-9 * ULINT_TO_LREAL(systime_ns));
  preSysTime := SysTime;
  tmpCycle := ULINT_TO_LREAL(systime_s - preSys_s) + 1.0E-9 * (ULINT_TO_LREAL(systime_ns) - ULINT_TO_LREAL(preSys_ns));
  cur_Cycle := LREAL_TO_REAL(tmpCycle);
  preSys_s := systime_s;
  preSys_ns := systime_ns;
  IF gStart_Tmr < 99999.9 THEN gStart_Tmr := gStart_Tmr + cur_Cycle; END_IF;
  Timings();

  IF  _init (*or external_init_ai *) then           (* Требуется инициализация структур и ФБ. *)
    (* Инициализация аналоговых входов. *)
      AI_structs_ini(init := TRUE);
      AI_Proc((*init := FALSE*));

    (* Инициализация дискретных входов. *)
      DI_structs_ini(init := TRUE);
      DI_Proc((*init := FALSE*));

      (* Инициализация аналоговых выходов. *)
  (*     AO_structs_ini(init := TRUE);
         AO_Proc(init := TRUE);*)

    (* Инициализация дискретных выходов. *)
      DO_structs_ini(init := TRUE);
      DO_Proc((*init := FALSE*));

     (* Инициализация ИМ. *)
      IM_structs_ini(init := TRUE);
      IM_Proc();

     (* Инициализация Защит *)
      Protections_structs_ini(init := TRUE);
      (*Protections_Proc();*)

       (* Стартовая инициализация OPC-тэгов элементами канальных структур. *)
          (*___________________AI______________________________________________________________________________*)
      (*ini_AI_OPC();*)

      _init := FALSE;

    ELSE                         (* Завершена инициализация структур и ФБ. *)

  (* Перенос OPC-тэгов в элементы структур каналов. *)
        (*___________________________________________AI________________________________________________*)
      (*Get_AI_OPC(); *)
       Get_algoritms_OPC();

     (* Пересчёт защит САУ. *)
     ProtectionsManager(protectManager);

       (* Пересчёт алгоритмов САУ. *)
     AlgoritmsManager(algManager);

      (****               Опрос входов.              ****)
          (* Опрос аналоговых входов. *)
      AI_Proc((*init := FALSE*));

          (* Опрос дискретных входов. *)
      DI_Proc((*init := FALSE*));

      (****              Запись выходов.             ****)
          (* Запись аналоговых выходов. *)
  (*    AO_Proc(init := FALSE);*)

       (* Запись дискретных выходов. *)
      DO_Proc((*init := FALSE*));

      (****               Опрос ИМ              ****)
      IM_Proc();

      (****            Опрос Защит              ****)
      Protections_Proc();

      Algoritms_Proc();

  END_IF;

  (* Передача информации на верхний уровень по OPC UA протоколу. *)
    (* Передача состояний каналов AI. *)
  (*Set_AI_OPC();)*
  (* Передача состояний каналов ИМ. *)
  (* Передача состояний защит. *)
  (* Передача состояний алгоритмов. *)
  Set_algoritms_OPC();
END_PROGRAM

CONFIGURATION config1
  VAR_GLOBAL
    systime_s AT %IL0.10.10 : ULINT;
    systime_ns AT %IL0.10.11 : ULINT;
    current_retrieve_us AT %IL0.10.12 : ULINT;
    current_config_us AT %IL0.10.13 : ULINT;
    current_publish_us AT %IL0.10.14 : ULINT;
    current_run_us AT %IL0.10.15 : ULINT;
    max_retrieve_us AT %QL0.10.16 : ULINT;
    max_config_us AT %QL0.10.17 : ULINT;
    max_publish_us AT %QL0.10.18 : ULINT;
    plc_run_number AT %IL0.10.19 : ULINT;
    arAIN_0 : TItemAIN;
    arAIN_1 : TItemAIN;
    arAIN_2 : TItemAIN;
    arAIN_3 : TItemAIN;
    arAIN_4 : TItemAIN;
    arAIN_5 : TItemAIN;
    arAIN_6 : TItemAIN;
    arAIN_7 : TItemAIN;
    arAIN_8 : TItemAIN;
    arAIN_9 : TItemAIN;
    arAIN_10 : TItemAIN;
    arAIN_11 : TItemAIN;
    arAIN_12 : TItemAIN;
    arAIN_13 : TItemAIN;
    arAIN_14 : TItemAIN;
    arAIN_15 : TItemAIN;
    arAIN_16 : TItemAIN;
    arAIN_17 : TItemAIN;
    arAIN_18 : TItemAIN;
    arAIN_19 : TItemAIN;
    arAIN_20 : TItemAIN;
    arAIN_21 : TItemAIN;
    arAIN_22 : TItemAIN;
    arAIN_23 : TItemAIN;
    arAIN_24 : TItemAIN;
    arAIN_25 : TItemAIN;
    arAIN_26 : TItemAIN;
    arAIN_27 : TItemAIN;
    arAIN_28 : TItemAIN;
    arAIN_29 : TItemAIN;
    arAIN_30 : TItemAIN;
    arAIN_31 : TItemAIN;
    arAIN_32 : TItemAIN;
    arAIN_33 : TItemAIN;
    arAIN_34 : TItemAIN;
    arAIN_35 : TItemAIN;
    arAIN_36 : TItemAIN;
    arAIN_37 : TItemAIN;
    arAIN_38 : TItemAIN;
    arAIN_39 : TItemAIN;
    arAIN_40 : TItemAIN;
    arAIN_41 : TItemAIN;
    arAIN_42 : TItemAIN;
    arAIN_43 : TItemAIN;
    arAIN_44 : TItemAIN;
    arAIN_45 : TItemAIN;
    arAIN_46 : TItemAIN;
    arAIN_47 : TItemAIN;
    arAIN_48 : TItemAIN;
    arAIN_49 : TItemAIN;
    arAIN_50 : TItemAIN;
    arAIN_51 : TItemAIN;
    arAIN_52 : TItemAIN;
    arAIN_53 : TItemAIN;
    arAIN_54 : TItemAIN;
    arAIN_55 : TItemAIN;
    arAIN_56 : TItemAIN;
    arAIN_57 : TItemAIN;
    arAIN_58 : TItemAIN;
    arAIN_59 : TItemAIN;
    arAIN_60 : TItemAIN;
    arAIN_61 : TItemAIN;
    arAIN_62 : TItemAIN;
    arAIN_63 : TItemAIN;
    arAIN_64 : TItemAIN;
    arAIN_65 : TItemAIN;
    arAIN_66 : TItemAIN;
    arAIN_67 : TItemAIN;
    arAIN_68 : TItemAIN;
    arAIN_69 : TItemAIN;
    arAIN_70 : TItemAIN;
    arAIN_71 : TItemAIN;
    arAIN_72 : TItemAIN;
    arAIN_73 : TItemAIN;
    arAIN_74 : TItemAIN;
    arAIN_75 : TItemAIN;
    arAIN_76 : TItemAIN;
    arAIN_77 : TItemAIN;
    arAIN_78 : TItemAIN;
    arAIN_79 : TItemAIN;
    arDIN_0 : TItemDIN;
    arDIN_1 : TItemDIN;
    arDIN_2 : TItemDIN;
    arDIN_3 : TItemDIN;
    arDIN_4 : TItemDIN;
    arDIN_5 : TItemDIN;
    arDIN_6 : TItemDIN;
    arDIN_7 : TItemDIN;
    arDIN_8 : TItemDIN;
    arDIN_9 : TItemDIN;
    arDIN_10 : TItemDIN;
    arDIN_11 : TItemDIN;
    arDIN_12 : TItemDIN;
    arDIN_13 : TItemDIN;
    arDIN_14 : TItemDIN;
    arDIN_15 : TItemDIN;
    arDIN_16 : TItemDIN;
    arDIN_17 : TItemDIN;
    arDIN_18 : TItemDIN;
    arDIN_19 : TItemDIN;
    arDIN_20 : TItemDIN;
    arDIN_21 : TItemDIN;
    arAOUT_0 : TDoubleData;
    arAOUT_1 : TDoubleData;
    arDOUT_0 : TWordData;
    arDOUT_1 : TWordData;
    arDOUT_2 : TWordData;
    arDOUT_3 : TWordData;
    arDOUT_4 : TWordData;
    arDOUT_66 : TWordData;
    arERR_0 : TItemDIN;
    arERR_1 : TItemDIN;
    arERR_2 : TItemDIN;
    arERR_3 : TItemDIN;
    arERR_4 : TItemDIN;
    arERR_5 : TItemDIN;
    arERR_6 : TItemDIN;
    arERR_7 : TItemDIN;
    arERR_8 : TItemDIN;
    arERR_9 : TItemDIN;
    arERR_10 : TItemDIN;
    arERR_11 : TItemDIN;
    arERR_12 : TItemDIN;
    arERR_13 : TItemDIN;
    arERR_14 : TItemDIN;
    arERR_15 : TItemDIN;
    arERR_16 : TItemDIN;
    arERR_17 : TItemDIN;
    arERR_18 : TItemDIN;
    arERR_19 : TItemDIN;
    arERR_20 : TItemDIN;
    arERR_21 : TItemDIN;
    arERR_22 : TItemDIN;
    arERR_23 : TItemDIN;
    arERR_24 : TItemDIN;
    arERR_66 : TItemDIN;
    arRelSt_0 : TItemDIN;
  END_VAR

  RESOURCE resource1 ON PLC
    VAR_GLOBAL CONSTANT
      gMaint_Time : REAL;
    END_VAR
    VAR_GLOBAL
      cur_Cycle : REAL;
      gStart_Tmr : REAL;
    END_VAR
    VAR_GLOBAL CONSTANT
      req_Cycle : REAL := 0.02;
    END_VAR
    VAR_GLOBAL
      gF_T_100mSec : BOOL;
      gT_1Sec : BOOL;
      gF_T_1Sec : BOOL;
      gT_1Min : BOOL;
      gR_T_1Min : BOOL;
      gF_T_1Min : BOOL;
      T_1SEC : REAL;
      del_T : REAL;
      ai : AiConfig;
      di : DiConfig;
      od : DOconfig;
      ao : AOConfig;
      IM : ImConfig;
      protections : ProtectionsConfig;
      algoritms : AlgoritmsConfig;
      algManager : struct_AlgoritmsManager;
      ModeGpa : TYPE_ModeGpa;
      protectManager : struct_ProtectionsManager;
      NotHasRezervNU : BOOL;
      Reset_HasNU : BOOL;
      AlgTimers : struct_AlgTimers;
      AlgQuestions : AlgoritmsQuestions;
      PMcommand : TYPE_CommandsPotectionsManager;
      AI_Kontrol_per_220V_HL AT %QL0.927 : LREAL;
      AI_Kontrol_per_220V_HW AT %QL0.934 : LREAL;
      AI_Kontrol_per_220V_LL AT %QL0.928 : LREAL;
      AI_Kontrol_per_220V_LW AT %QL0.936 : LREAL;
      AI_Kontrol_per_220V_command AT %QW0.931 : UINT;
      AI_Kontrol_per_220V_newHL AT %QL0.929 : LREAL;
      AI_Kontrol_per_220V_newHW AT %QL0.935 : LREAL;
      AI_Kontrol_per_220V_newLL AT %QL0.930 : LREAL;
      AI_Kontrol_per_220V_newLW AT %QL0.937 : LREAL;
      AI_Kontrol_per_220V_status AT %QD0.932 : UDINT;
      AI_Kontrol_per_220V_value AT %QL0.933 : LREAL;
      AI_Kontrol_post_220V_HL AT %QL0.938 : LREAL;
      AI_Kontrol_post_220V_HW AT %QL0.945 : LREAL;
      AI_Kontrol_post_220V_LL AT %QL0.939 : LREAL;
      AI_Kontrol_post_220V_LW AT %QL0.947 : LREAL;
      AI_Kontrol_post_220V_command AT %QW0.942 : UINT;
      AI_Kontrol_post_220V_newHL AT %QL0.940 : LREAL;
      AI_Kontrol_post_220V_newHW AT %QL0.946 : LREAL;
      AI_Kontrol_post_220V_newLL AT %QL0.941 : LREAL;
      AI_Kontrol_post_220V_newLW AT %QL0.948 : LREAL;
      AI_Kontrol_post_220V_status AT %QD0.943 : UDINT;
      AI_Kontrol_post_220V_value AT %QL0.944 : LREAL;
      AI_Os_sdvig_nagnetatelja_minus_HL AT %QL0.864 : LREAL;
      AI_Os_sdvig_nagnetatelja_minus_LA AT %QL0.873 : LREAL;
      AI_Os_sdvig_nagnetatelja_minus_LL AT %QL0.865 : LREAL;
      AI_Os_sdvig_nagnetatelja_minus_LW AT %QL0.871 : LREAL;
      AI_Os_sdvig_nagnetatelja_minus_command AT %QW0.868 : UINT;
      AI_Os_sdvig_nagnetatelja_minus_newHL AT %QL0.866 : LREAL;
      AI_Os_sdvig_nagnetatelja_minus_newLA AT %QL0.874 : LREAL;
      AI_Os_sdvig_nagnetatelja_minus_newLL AT %QL0.867 : LREAL;
      AI_Os_sdvig_nagnetatelja_minus_newLW AT %QL0.872 : LREAL;
      AI_Os_sdvig_nagnetatelja_minus_status AT %QD0.869 : UDINT;
      AI_Os_sdvig_nagnetatelja_minus_value AT %QL0.870 : LREAL;
      AI_Os_sdvig_nagnetatelja_plus_HA AT %QL0.426 : LREAL;
      AI_Os_sdvig_nagnetatelja_plus_HL AT %QL0.417 : LREAL;
      AI_Os_sdvig_nagnetatelja_plus_HW AT %QL0.424 : LREAL;
      AI_Os_sdvig_nagnetatelja_plus_LL AT %QL0.418 : LREAL;
      AI_Os_sdvig_nagnetatelja_plus_command AT %QW0.421 : UINT;
      AI_Os_sdvig_nagnetatelja_plus_newHA AT %QL0.863 : LREAL;
      AI_Os_sdvig_nagnetatelja_plus_newHL AT %QL0.419 : LREAL;
      AI_Os_sdvig_nagnetatelja_plus_newHW AT %QL0.425 : LREAL;
      AI_Os_sdvig_nagnetatelja_plus_newLL AT %QL0.420 : LREAL;
      AI_Os_sdvig_nagnetatelja_plus_status AT %QD0.422 : UDINT;
      AI_Os_sdvig_nagnetatelja_plus_value AT %QL0.423 : LREAL;
      AI_Pgaza_na_vhode_nagnetatelia_HL AT %QL0.359 : LREAL;
      AI_Pgaza_na_vhode_nagnetatelia_LL AT %QL0.360 : LREAL;
      AI_Pgaza_na_vhode_nagnetatelia_LW AT %QL0.366 : LREAL;
      AI_Pgaza_na_vhode_nagnetatelia_command AT %QW0.363 : UINT;
      AI_Pgaza_na_vhode_nagnetatelia_newHL AT %QL0.361 : LREAL;
      AI_Pgaza_na_vhode_nagnetatelia_newLL AT %QL0.362 : LREAL;
      AI_Pgaza_na_vhode_nagnetatelia_newLW AT %QL0.367 : LREAL;
      AI_Pgaza_na_vhode_nagnetatelia_status AT %QD0.364 : UDINT;
      AI_Pgaza_na_vhode_nagnetatelia_value AT %QL0.365 : LREAL;
      AI_Pgaza_na_vyhode_nagnetatelia_HA AT %QL0.377 : LREAL;
      AI_Pgaza_na_vyhode_nagnetatelia_HL AT %QL0.368 : LREAL;
      AI_Pgaza_na_vyhode_nagnetatelia_LL AT %QL0.369 : LREAL;
      AI_Pgaza_na_vyhode_nagnetatelia_LW AT %QL0.375 : LREAL;
      AI_Pgaza_na_vyhode_nagnetatelia_command AT %QW0.372 : UINT;
      AI_Pgaza_na_vyhode_nagnetatelia_newHA AT %QL0.378 : LREAL;
      AI_Pgaza_na_vyhode_nagnetatelia_newHL AT %QL0.370 : LREAL;
      AI_Pgaza_na_vyhode_nagnetatelia_newLL AT %QL0.371 : LREAL;
      AI_Pgaza_na_vyhode_nagnetatelia_newLW AT %QL0.376 : LREAL;
      AI_Pgaza_na_vyhode_nagnetatelia_status AT %QD0.373 : UDINT;
      AI_Pgaza_na_vyhode_nagnetatelia_value AT %QL0.374 : LREAL;
      AI_Pimpuls_gaz_HL AT %QL0.379 : LREAL;
      AI_Pimpuls_gaz_LL AT %QL0.380 : LREAL;
      AI_Pimpuls_gaz_LW AT %QL0.386 : LREAL;
      AI_Pimpuls_gaz_command AT %QW0.383 : UINT;
      AI_Pimpuls_gaz_newHL AT %QL0.381 : LREAL;
      AI_Pimpuls_gaz_newLL AT %QL0.382 : LREAL;
      AI_Pimpuls_gaz_newLW AT %QL0.387 : LREAL;
      AI_Pimpuls_gaz_status AT %QD0.384 : UDINT;
      AI_Pimpuls_gaz_value AT %QL0.385 : LREAL;
      AI_Pmasla_posle_GNS_HL AT %QL0.339 : LREAL;
      AI_Pmasla_posle_GNS_HW AT %QL0.346 : LREAL;
      AI_Pmasla_posle_GNS_LL AT %QL0.340 : LREAL;
      AI_Pmasla_posle_GNS_LW AT %QL0.348 : LREAL;
      AI_Pmasla_posle_GNS_command AT %QW0.343 : UINT;
      AI_Pmasla_posle_GNS_newHL AT %QL0.341 : LREAL;
      AI_Pmasla_posle_GNS_newHW AT %QL0.347 : LREAL;
      AI_Pmasla_posle_GNS_newLL AT %QL0.342 : LREAL;
      AI_Pmasla_posle_GNS_newLW AT %QL0.349 : LREAL;
      AI_Pmasla_posle_GNS_status AT %QD0.344 : UDINT;
      AI_Pmasla_posle_GNS_value AT %QL0.345 : LREAL;
      AI_Pmasla_posle_NU_HL AT %QL0.350 : LREAL;
      AI_Pmasla_posle_NU_LL AT %QL0.351 : LREAL;
      AI_Pmasla_posle_NU_LW AT %QL0.357 : LREAL;
      AI_Pmasla_posle_NU_command AT %QW0.354 : UINT;
      AI_Pmasla_posle_NU_newHL AT %QL0.352 : LREAL;
      AI_Pmasla_posle_NU_newLL AT %QL0.353 : LREAL;
      AI_Pmasla_posle_NU_newLW AT %QL0.358 : LREAL;
      AI_Pmasla_posle_NU_status AT %QD0.355 : UDINT;
      AI_Pmasla_posle_NU_value AT %QL0.356 : LREAL;
      AI_Pmaslo_sm_nizkoe_HL AT %QL0.317 : LREAL;
      AI_Pmaslo_sm_nizkoe_LA AT %QL0.326 : LREAL;
      AI_Pmaslo_sm_nizkoe_LL AT %QL0.318 : LREAL;
      AI_Pmaslo_sm_nizkoe_LW AT %QL0.324 : LREAL;
      AI_Pmaslo_sm_nizkoe_command AT %QW0.321 : UINT;
      AI_Pmaslo_sm_nizkoe_newHL AT %QL0.319 : LREAL;
      AI_Pmaslo_sm_nizkoe_newLA AT %QL0.327 : LREAL;
      AI_Pmaslo_sm_nizkoe_newLL AT %QL0.320 : LREAL;
      AI_Pmaslo_sm_nizkoe_newLW AT %QL0.325 : LREAL;
      AI_Pmaslo_sm_nizkoe_status AT %QD0.322 : UDINT;
      AI_Pmaslo_sm_nizkoe_value AT %QL0.323 : LREAL;
      AI_Pmaslo_sm_vysokoe_HL AT %QL0.328 : LREAL;
      AI_Pmaslo_sm_vysokoe_LA AT %QL0.337 : LREAL;
      AI_Pmaslo_sm_vysokoe_LL AT %QL0.329 : LREAL;
      AI_Pmaslo_sm_vysokoe_LW AT %QL0.335 : LREAL;
      AI_Pmaslo_sm_vysokoe_command AT %QW0.332 : UINT;
      AI_Pmaslo_sm_vysokoe_newHL AT %QL0.330 : LREAL;
      AI_Pmaslo_sm_vysokoe_newLA AT %QL0.338 : LREAL;
      AI_Pmaslo_sm_vysokoe_newLL AT %QL0.331 : LREAL;
      AI_Pmaslo_sm_vysokoe_newLW AT %QL0.336 : LREAL;
      AI_Pmaslo_sm_vysokoe_status AT %QD0.333 : UDINT;
      AI_Pmaslo_sm_vysokoe_value AT %QL0.334 : LREAL;
      AI_Tgaza_na_vhode_H_HL AT %QL0.254 : LREAL;
      AI_Tgaza_na_vhode_H_HW AT %QL0.261 : LREAL;
      AI_Tgaza_na_vhode_H_LL AT %QL0.255 : LREAL;
      AI_Tgaza_na_vhode_H_command AT %QW0.258 : UINT;
      AI_Tgaza_na_vhode_H_newHL AT %QL0.256 : LREAL;
      AI_Tgaza_na_vhode_H_newHW AT %QL0.262 : LREAL;
      AI_Tgaza_na_vhode_H_newLL AT %QL0.257 : LREAL;
      AI_Tgaza_na_vhode_H_status AT %QD0.259 : UDINT;
      AI_Tgaza_na_vhode_H_value AT %QL0.260 : LREAL;
      AI_Tgaza_na_vyhode_H_HA AT %QL0.272 : LREAL;
      AI_Tgaza_na_vyhode_H_HL AT %QL0.263 : LREAL;
      AI_Tgaza_na_vyhode_H_HW AT %QL0.270 : LREAL;
      AI_Tgaza_na_vyhode_H_LL AT %QL0.264 : LREAL;
      AI_Tgaza_na_vyhode_H_command AT %QW0.267 : UINT;
      AI_Tgaza_na_vyhode_H_newHA AT %QL0.273 : LREAL;
      AI_Tgaza_na_vyhode_H_newHL AT %QL0.265 : LREAL;
      AI_Tgaza_na_vyhode_H_newHW AT %QL0.271 : LREAL;
      AI_Tgaza_na_vyhode_H_newLL AT %QL0.266 : LREAL;
      AI_Tgaza_na_vyhode_H_status AT %QD0.268 : UDINT;
      AI_Tgaza_na_vyhode_H_value AT %QL0.269 : LREAL;
      AI_Tgorjachego_vozduha_ED_kanal_1_HL AT %QL0.227 : LREAL;
      AI_Tgorjachego_vozduha_ED_kanal_1_HW AT %QL0.234 : LREAL;
      AI_Tgorjachego_vozduha_ED_kanal_1_LL AT %QL0.228 : LREAL;
      AI_Tgorjachego_vozduha_ED_kanal_1_command AT %QW0.231 : UINT;
      AI_Tgorjachego_vozduha_ED_kanal_1_newHL AT %QL0.229 : LREAL;
      AI_Tgorjachego_vozduha_ED_kanal_1_newHW AT %QL0.235 : LREAL;
      AI_Tgorjachego_vozduha_ED_kanal_1_newLL AT %QL0.230 : LREAL;
      AI_Tgorjachego_vozduha_ED_kanal_1_status AT %QD0.232 : UDINT;
      AI_Tgorjachego_vozduha_ED_kanal_1_value AT %QL0.233 : LREAL;
      AI_Tgorjachego_vozduha_ED_kanal_2_HL AT %QL0.236 : LREAL;
      AI_Tgorjachego_vozduha_ED_kanal_2_HW AT %QL0.243 : LREAL;
      AI_Tgorjachego_vozduha_ED_kanal_2_LL AT %QL0.237 : LREAL;
      AI_Tgorjachego_vozduha_ED_kanal_2_command AT %QW0.240 : UINT;
      AI_Tgorjachego_vozduha_ED_kanal_2_newHL AT %QL0.238 : LREAL;
      AI_Tgorjachego_vozduha_ED_kanal_2_newHW AT %QL0.244 : LREAL;
      AI_Tgorjachego_vozduha_ED_kanal_2_newLL AT %QL0.239 : LREAL;
      AI_Tgorjachego_vozduha_ED_kanal_2_status AT %QD0.241 : UDINT;
      AI_Tgorjachego_vozduha_ED_kanal_2_value AT %QL0.242 : LREAL;
      AI_Tholodnogo_vozduha_ED_kanal_1_HL AT %QL0.209 : LREAL;
      AI_Tholodnogo_vozduha_ED_kanal_1_HW AT %QL0.216 : LREAL;
      AI_Tholodnogo_vozduha_ED_kanal_1_LL AT %QL0.210 : LREAL;
      AI_Tholodnogo_vozduha_ED_kanal_1_command AT %QW0.213 : UINT;
      AI_Tholodnogo_vozduha_ED_kanal_1_newHL AT %QL0.211 : LREAL;
      AI_Tholodnogo_vozduha_ED_kanal_1_newHW AT %QL0.217 : LREAL;
      AI_Tholodnogo_vozduha_ED_kanal_1_newLL AT %QL0.212 : LREAL;
      AI_Tholodnogo_vozduha_ED_kanal_1_status AT %QD0.214 : UDINT;
      AI_Tholodnogo_vozduha_ED_kanal_1_value AT %QL0.215 : LREAL;
      AI_Tholodnogo_vozduha_ED_kanal_2_HL AT %QL0.218 : LREAL;
      AI_Tholodnogo_vozduha_ED_kanal_2_HW AT %QL0.225 : LREAL;
      AI_Tholodnogo_vozduha_ED_kanal_2_LL AT %QL0.219 : LREAL;
      AI_Tholodnogo_vozduha_ED_kanal_2_command AT %QW0.222 : UINT;
      AI_Tholodnogo_vozduha_ED_kanal_2_newHL AT %QL0.220 : LREAL;
      AI_Tholodnogo_vozduha_ED_kanal_2_newHW AT %QL0.226 : LREAL;
      AI_Tholodnogo_vozduha_ED_kanal_2_newLL AT %QL0.221 : LREAL;
      AI_Tholodnogo_vozduha_ED_kanal_2_status AT %QD0.223 : UDINT;
      AI_Tholodnogo_vozduha_ED_kanal_2_value AT %QL0.224 : LREAL;
      AI_Tmasla_MB_HL AT %QL0.292 : LREAL;
      AI_Tmasla_MB_HW AT %QL0.299 : LREAL;
      AI_Tmasla_MB_LL AT %QL0.293 : LREAL;
      AI_Tmasla_MB_TEN_HL AT %QL0.301 : LREAL;
      AI_Tmasla_MB_TEN_HW AT %QL0.308 : LREAL;
      AI_Tmasla_MB_TEN_LL AT %QL0.302 : LREAL;
      AI_Tmasla_MB_TEN_command AT %QW0.305 : UINT;
      AI_Tmasla_MB_TEN_newHL AT %QL0.303 : LREAL;
      AI_Tmasla_MB_TEN_newHW AT %QL0.309 : LREAL;
      AI_Tmasla_MB_TEN_newLL AT %QL0.304 : LREAL;
      AI_Tmasla_MB_TEN_status AT %QD0.306 : UDINT;
      AI_Tmasla_MB_TEN_value AT %QL0.307 : LREAL;
      AI_Tmasla_MB_command AT %QW0.296 : UINT;
      AI_Tmasla_MB_newHL AT %QL0.294 : LREAL;
      AI_Tmasla_MB_newHW AT %QL0.300 : LREAL;
      AI_Tmasla_MB_newLL AT %QL0.295 : LREAL;
      AI_Tmasla_MB_status AT %QD0.297 : UDINT;
      AI_Tmasla_MB_value AT %QL0.298 : LREAL;
      AI_Tmasla_do_AVOM_HL AT %QL0.274 : LREAL;
      AI_Tmasla_do_AVOM_HW AT %QL0.281 : LREAL;
      AI_Tmasla_do_AVOM_LL AT %QL0.275 : LREAL;
      AI_Tmasla_do_AVOM_command AT %QW0.278 : UINT;
      AI_Tmasla_do_AVOM_newHL AT %QL0.276 : LREAL;
      AI_Tmasla_do_AVOM_newHW AT %QL0.282 : LREAL;
      AI_Tmasla_do_AVOM_newLL AT %QL0.277 : LREAL;
      AI_Tmasla_do_AVOM_status AT %QD0.279 : UDINT;
      AI_Tmasla_do_AVOM_value AT %QL0.280 : LREAL;
      AI_Tmasla_posle_AVOM_HL AT %QL0.283 : LREAL;
      AI_Tmasla_posle_AVOM_HW AT %QL0.290 : LREAL;
      AI_Tmasla_posle_AVOM_LL AT %QL0.284 : LREAL;
      AI_Tmasla_posle_AVOM_command AT %QW0.287 : UINT;
      AI_Tmasla_posle_AVOM_newHL AT %QL0.285 : LREAL;
      AI_Tmasla_posle_AVOM_newHW AT %QL0.291 : LREAL;
      AI_Tmasla_posle_AVOM_newLL AT %QL0.286 : LREAL;
      AI_Tmasla_posle_AVOM_status AT %QD0.288 : UDINT;
      AI_Tmasla_posle_AVOM_value AT %QL0.289 : LREAL;
      AI_Tmedi_statora_kanal_1_HL AT %QL0.28 : LREAL;
      AI_Tmedi_statora_kanal_1_HW AT %QL0.35 : LREAL;
      AI_Tmedi_statora_kanal_1_LL AT %QL0.29 : LREAL;
      AI_Tmedi_statora_kanal_1_command AT %QW0.32 : UINT;
      AI_Tmedi_statora_kanal_1_newHL AT %QL0.30 : LREAL;
      AI_Tmedi_statora_kanal_1_newHW AT %QL0.36 : LREAL;
      AI_Tmedi_statora_kanal_1_newLL AT %QL0.31 : LREAL;
      AI_Tmedi_statora_kanal_1_status AT %QD0.33 : UDINT;
      AI_Tmedi_statora_kanal_1_value AT %QL0.34 : LREAL;
      AI_Tmedi_statora_kanal_2_HL AT %QL0.37 : LREAL;
      AI_Tmedi_statora_kanal_2_HW AT %QL0.44 : LREAL;
      AI_Tmedi_statora_kanal_2_LL AT %QL0.38 : LREAL;
      AI_Tmedi_statora_kanal_2_command AT %QW0.41 : UINT;
      AI_Tmedi_statora_kanal_2_newHL AT %QL0.39 : LREAL;
      AI_Tmedi_statora_kanal_2_newHW AT %QL0.45 : LREAL;
      AI_Tmedi_statora_kanal_2_newLL AT %QL0.40 : LREAL;
      AI_Tmedi_statora_kanal_2_status AT %QD0.42 : UDINT;
      AI_Tmedi_statora_kanal_2_value AT %QL0.43 : LREAL;
      AI_Tmedi_statora_kanal_3_HL AT %QL0.46 : LREAL;
      AI_Tmedi_statora_kanal_3_HW AT %QL0.53 : LREAL;
      AI_Tmedi_statora_kanal_3_LL AT %QL0.47 : LREAL;
      AI_Tmedi_statora_kanal_3_command AT %QW0.50 : UINT;
      AI_Tmedi_statora_kanal_3_newHL AT %QL0.48 : LREAL;
      AI_Tmedi_statora_kanal_3_newHW AT %QL0.54 : LREAL;
      AI_Tmedi_statora_kanal_3_newLL AT %QL0.49 : LREAL;
      AI_Tmedi_statora_kanal_3_status AT %QD0.51 : UDINT;
      AI_Tmedi_statora_kanal_3_value AT %QL0.52 : LREAL;
      AI_Tnarujnogo_vozduha_HL AT %QL0.245 : LREAL;
      AI_Tnarujnogo_vozduha_HW AT %QL0.252 : LREAL;
      AI_Tnarujnogo_vozduha_LL AT %QL0.246 : LREAL;
      AI_Tnarujnogo_vozduha_command AT %QW0.249 : UINT;
      AI_Tnarujnogo_vozduha_newHL AT %QL0.247 : LREAL;
      AI_Tnarujnogo_vozduha_newHW AT %QL0.253 : LREAL;
      AI_Tnarujnogo_vozduha_newLL AT %QL0.248 : LREAL;
      AI_Tnarujnogo_vozduha_status AT %QD0.250 : UDINT;
      AI_Tnarujnogo_vozduha_value AT %QL0.251 : LREAL;
      AI_Tok_statora_HL AT %QL0.949 : LREAL;
      AI_Tok_statora_LL AT %QL0.950 : LREAL;
      AI_Tok_statora_LW AT %QL0.956 : LREAL;
      AI_Tok_statora_command AT %QW0.953 : UINT;
      AI_Tok_statora_newHL AT %QL0.951 : LREAL;
      AI_Tok_statora_newLL AT %QL0.952 : LREAL;
      AI_Tok_statora_newLW AT %QL0.957 : LREAL;
      AI_Tok_statora_status AT %QD0.954 : UDINT;
      AI_Tok_statora_value AT %QL0.955 : LREAL;
      AI_Toporno_podshipnika_EDT_1_HA AT %QL0.64 : LREAL;
      AI_Toporno_podshipnika_EDT_1_HL AT %QL0.55 : LREAL;
      AI_Toporno_podshipnika_EDT_1_HW AT %QL0.62 : LREAL;
      AI_Toporno_podshipnika_EDT_1_LL AT %QL0.56 : LREAL;
      AI_Toporno_podshipnika_EDT_1_command AT %QW0.59 : UINT;
      AI_Toporno_podshipnika_EDT_1_newHA AT %QL0.65 : LREAL;
      AI_Toporno_podshipnika_EDT_1_newHL AT %QL0.57 : LREAL;
      AI_Toporno_podshipnika_EDT_1_newHW AT %QL0.63 : LREAL;
      AI_Toporno_podshipnika_EDT_1_newLL AT %QL0.58 : LREAL;
      AI_Toporno_podshipnika_EDT_1_status AT %QD0.60 : UDINT;
      AI_Toporno_podshipnika_EDT_1_value AT %QL0.61 : LREAL;
      AI_Toy_podshipnika_EDT_2_HA AT %QL0.75 : LREAL;
      AI_Toy_podshipnika_EDT_2_HL AT %QL0.66 : LREAL;
      AI_Toy_podshipnika_EDT_2_HW AT %QL0.73 : LREAL;
      AI_Toy_podshipnika_EDT_2_LL AT %QL0.67 : LREAL;
      AI_Toy_podshipnika_EDT_2_command AT %QW0.70 : UINT;
      AI_Toy_podshipnika_EDT_2_newHA AT %QL0.76 : LREAL;
      AI_Toy_podshipnika_EDT_2_newHL AT %QL0.68 : LREAL;
      AI_Toy_podshipnika_EDT_2_newHW AT %QL0.74 : LREAL;
      AI_Toy_podshipnika_EDT_2_newLL AT %QL0.69 : LREAL;
      AI_Toy_podshipnika_EDT_2_status AT %QD0.71 : UDINT;
      AI_Toy_podshipnika_EDT_2_value AT %QL0.72 : LREAL;
      AI_Toy_podshipnika_kol_EDT_3_HA AT %QL0.86 : LREAL;
      AI_Toy_podshipnika_kol_EDT_3_HL AT %QL0.77 : LREAL;
      AI_Toy_podshipnika_kol_EDT_3_HW AT %QL0.84 : LREAL;
      AI_Toy_podshipnika_kol_EDT_3_LL AT %QL0.78 : LREAL;
      AI_Toy_podshipnika_kol_EDT_3_command AT %QW0.81 : UINT;
      AI_Toy_podshipnika_kol_EDT_3_newHA AT %QL0.87 : LREAL;
      AI_Toy_podshipnika_kol_EDT_3_newHL AT %QL0.79 : LREAL;
      AI_Toy_podshipnika_kol_EDT_3_newHW AT %QL0.85 : LREAL;
      AI_Toy_podshipnika_kol_EDT_3_newLL AT %QL0.80 : LREAL;
      AI_Toy_podshipnika_kol_EDT_3_status AT %QD0.82 : UDINT;
      AI_Toy_podshipnika_kol_EDT_3_value AT %QL0.83 : LREAL;
      AI_Toy_podshipnika_kol_EDT_4_HA AT %QL0.97 : LREAL;
      AI_Toy_podshipnika_kol_EDT_4_HL AT %QL0.88 : LREAL;
      AI_Toy_podshipnika_kol_EDT_4_HW AT %QL0.95 : LREAL;
      AI_Toy_podshipnika_kol_EDT_4_LL AT %QL0.89 : LREAL;
      AI_Toy_podshipnika_kol_EDT_4_command AT %QW0.92 : UINT;
      AI_Toy_podshipnika_kol_EDT_4_newHA AT %QL0.98 : LREAL;
      AI_Toy_podshipnika_kol_EDT_4_newHL AT %QL0.90 : LREAL;
      AI_Toy_podshipnika_kol_EDT_4_newHW AT %QL0.96 : LREAL;
      AI_Toy_podshipnika_kol_EDT_4_newLL AT %QL0.91 : LREAL;
      AI_Toy_podshipnika_kol_EDT_4_status AT %QD0.93 : UDINT;
      AI_Toy_podshipnika_kol_EDT_4_value AT %QL0.94 : LREAL;
      AI_Toy_podshipnika_nerab_kol_EDT_10_1_HA AT %QL0.196 : LREAL;
      AI_Toy_podshipnika_nerab_kol_EDT_10_1_HL AT %QL0.187 : LREAL;
      AI_Toy_podshipnika_nerab_kol_EDT_10_1_HW AT %QL0.194 : LREAL;
      AI_Toy_podshipnika_nerab_kol_EDT_10_1_LL AT %QL0.188 : LREAL;
      AI_Toy_podshipnika_nerab_kol_EDT_10_1_command AT %QW0.191 : UINT;
      AI_Toy_podshipnika_nerab_kol_EDT_10_1_newHA AT %QL0.197 : LREAL;
      AI_Toy_podshipnika_nerab_kol_EDT_10_1_newHL AT %QL0.189 : LREAL;
      AI_Toy_podshipnika_nerab_kol_EDT_10_1_newHW AT %QL0.195 : LREAL;
      AI_Toy_podshipnika_nerab_kol_EDT_10_1_newLL AT %QL0.190 : LREAL;
      AI_Toy_podshipnika_nerab_kol_EDT_10_1_status AT %QD0.192 : UDINT;
      AI_Toy_podshipnika_nerab_kol_EDT_10_1_value AT %QL0.193 : LREAL;
      AI_Toy_podshipnika_nerab_kol_EDT_10_2_HA AT %QL0.207 : LREAL;
      AI_Toy_podshipnika_nerab_kol_EDT_10_2_HL AT %QL0.198 : LREAL;
      AI_Toy_podshipnika_nerab_kol_EDT_10_2_HW AT %QL0.205 : LREAL;
      AI_Toy_podshipnika_nerab_kol_EDT_10_2_LL AT %QL0.199 : LREAL;
      AI_Toy_podshipnika_nerab_kol_EDT_10_2_command AT %QW0.202 : UINT;
      AI_Toy_podshipnika_nerab_kol_EDT_10_2_newHA AT %QL0.208 : LREAL;
      AI_Toy_podshipnika_nerab_kol_EDT_10_2_newHL AT %QL0.200 : LREAL;
      AI_Toy_podshipnika_nerab_kol_EDT_10_2_newHW AT %QL0.206 : LREAL;
      AI_Toy_podshipnika_nerab_kol_EDT_10_2_newLL AT %QL0.201 : LREAL;
      AI_Toy_podshipnika_nerab_kol_EDT_10_2_status AT %QD0.203 : UDINT;
      AI_Toy_podshipnika_nerab_kol_EDT_10_2_value AT %QL0.204 : LREAL;
      AI_Toy_podshipnika_rab_kol_EDT_9_1_HA AT %QL0.174 : LREAL;
      AI_Toy_podshipnika_rab_kol_EDT_9_1_HL AT %QL0.165 : LREAL;
      AI_Toy_podshipnika_rab_kol_EDT_9_1_HW AT %QL0.172 : LREAL;
      AI_Toy_podshipnika_rab_kol_EDT_9_1_LL AT %QL0.166 : LREAL;
      AI_Toy_podshipnika_rab_kol_EDT_9_1_command AT %QW0.169 : UINT;
      AI_Toy_podshipnika_rab_kol_EDT_9_1_newHA AT %QL0.175 : LREAL;
      AI_Toy_podshipnika_rab_kol_EDT_9_1_newHL AT %QL0.167 : LREAL;
      AI_Toy_podshipnika_rab_kol_EDT_9_1_newHW AT %QL0.173 : LREAL;
      AI_Toy_podshipnika_rab_kol_EDT_9_1_newLL AT %QL0.168 : LREAL;
      AI_Toy_podshipnika_rab_kol_EDT_9_1_status AT %QD0.170 : UDINT;
      AI_Toy_podshipnika_rab_kol_EDT_9_1_value AT %QL0.171 : LREAL;
      AI_Toy_podshipnika_rab_kol_EDT_9_2_HA AT %QL0.185 : LREAL;
      AI_Toy_podshipnika_rab_kol_EDT_9_2_HL AT %QL0.176 : LREAL;
      AI_Toy_podshipnika_rab_kol_EDT_9_2_HW AT %QL0.183 : LREAL;
      AI_Toy_podshipnika_rab_kol_EDT_9_2_LL AT %QL0.177 : LREAL;
      AI_Toy_podshipnika_rab_kol_EDT_9_2_command AT %QW0.180 : UINT;
      AI_Toy_podshipnika_rab_kol_EDT_9_2_newHA AT %QL0.186 : LREAL;
      AI_Toy_podshipnika_rab_kol_EDT_9_2_newHL AT %QL0.178 : LREAL;
      AI_Toy_podshipnika_rab_kol_EDT_9_2_newHW AT %QL0.184 : LREAL;
      AI_Toy_podshipnika_rab_kol_EDT_9_2_newLL AT %QL0.179 : LREAL;
      AI_Toy_podshipnika_rab_kol_EDT_9_2_status AT %QD0.181 : UDINT;
      AI_Toy_podshipnika_rab_kol_EDT_9_2_value AT %QL0.182 : LREAL;
      AI_Toy_podshipnika_shest_red_EDT_5_HA AT %QL0.108 : LREAL;
      AI_Toy_podshipnika_shest_red_EDT_5_HL AT %QL0.99 : LREAL;
      AI_Toy_podshipnika_shest_red_EDT_5_HW AT %QL0.106 : LREAL;
      AI_Toy_podshipnika_shest_red_EDT_5_LL AT %QL0.100 : LREAL;
      AI_Toy_podshipnika_shest_red_EDT_5_command AT %QW0.103 : UINT;
      AI_Toy_podshipnika_shest_red_EDT_5_newHA AT %QL0.109 : LREAL;
      AI_Toy_podshipnika_shest_red_EDT_5_newHL AT %QL0.101 : LREAL;
      AI_Toy_podshipnika_shest_red_EDT_5_newHW AT %QL0.107 : LREAL;
      AI_Toy_podshipnika_shest_red_EDT_5_newLL AT %QL0.102 : LREAL;
      AI_Toy_podshipnika_shest_red_EDT_5_status AT %QD0.104 : UDINT;
      AI_Toy_podshipnika_shest_red_EDT_5_value AT %QL0.105 : LREAL;
      AI_Toy_podshipnika_svobod_konca_EDT_8_1_HA AT %QL0.152 : LREAL;
      AI_Toy_podshipnika_svobod_konca_EDT_8_1_HL AT %QL0.143 : LREAL;
      AI_Toy_podshipnika_svobod_konca_EDT_8_1_HW AT %QL0.150 : LREAL;
      AI_Toy_podshipnika_svobod_konca_EDT_8_1_LL AT %QL0.144 : LREAL;
      AI_Toy_podshipnika_svobod_konca_EDT_8_1_command AT %QW0.147 : UINT;
      AI_Toy_podshipnika_svobod_konca_EDT_8_1_newHA AT %QL0.153 : LREAL;
      AI_Toy_podshipnika_svobod_konca_EDT_8_1_newHL AT %QL0.145 : LREAL;
      AI_Toy_podshipnika_svobod_konca_EDT_8_1_newHW AT %QL0.151 : LREAL;
      AI_Toy_podshipnika_svobod_konca_EDT_8_1_newLL AT %QL0.146 : LREAL;
      AI_Toy_podshipnika_svobod_konca_EDT_8_1_status AT %QD0.148 : UDINT;
      AI_Toy_podshipnika_svobod_konca_EDT_8_1_value AT %QL0.149 : LREAL;
      AI_Toy_podshipnika_svobod_konca_EDT_8_2_HA AT %QL0.163 : LREAL;
      AI_Toy_podshipnika_svobod_konca_EDT_8_2_HL AT %QL0.154 : LREAL;
      AI_Toy_podshipnika_svobod_konca_EDT_8_2_HW AT %QL0.161 : LREAL;
      AI_Toy_podshipnika_svobod_konca_EDT_8_2_LL AT %QL0.155 : LREAL;
      AI_Toy_podshipnika_svobod_konca_EDT_8_2_command AT %QW0.158 : UINT;
      AI_Toy_podshipnika_svobod_konca_EDT_8_2_newHA AT %QL0.164 : LREAL;
      AI_Toy_podshipnika_svobod_konca_EDT_8_2_newHL AT %QL0.156 : LREAL;
      AI_Toy_podshipnika_svobod_konca_EDT_8_2_newHW AT %QL0.162 : LREAL;
      AI_Toy_podshipnika_svobod_konca_EDT_8_2_newLL AT %QL0.157 : LREAL;
      AI_Toy_podshipnika_svobod_konca_EDT_8_2_status AT %QD0.159 : UDINT;
      AI_Toy_podshipnika_svobod_konca_EDT_8_2_value AT %QL0.160 : LREAL;
      AI_Tshu_HL AT %QL0.310 : LREAL;
      AI_Tshu_LL AT %QL0.311 : LREAL;
      AI_Tshu_command AT %QW0.314 : UINT;
      AI_Tshu_newHL AT %QL0.312 : LREAL;
      AI_Tshu_newLL AT %QL0.313 : LREAL;
      AI_Tshu_status AT %QD0.315 : UDINT;
      AI_Tshu_value AT %QL0.316 : LREAL;
      AI_Tstali_statora_kanal_1_HL AT %QL0.1 : LREAL;
      AI_Tstali_statora_kanal_1_HW AT %QL0.8 : LREAL;
      AI_Tstali_statora_kanal_1_LL AT %QL0.2 : LREAL;
      AI_Tstali_statora_kanal_1_command AT %QW0.5 : UINT;
      AI_Tstali_statora_kanal_1_newHL AT %QL0.3 : LREAL;
      AI_Tstali_statora_kanal_1_newHW AT %QL0.9 : LREAL;
      AI_Tstali_statora_kanal_1_newLL AT %QL0.4 : LREAL;
      AI_Tstali_statora_kanal_1_status AT %QD0.6 : UDINT;
      AI_Tstali_statora_kanal_1_value AT %QL0.7 : LREAL;
      AI_Tstali_statora_kanal_2_HL AT %QL0.10 : LREAL;
      AI_Tstali_statora_kanal_2_HW AT %QL0.17 : LREAL;
      AI_Tstali_statora_kanal_2_LL AT %QL0.11 : LREAL;
      AI_Tstali_statora_kanal_2_command AT %QW0.14 : UINT;
      AI_Tstali_statora_kanal_2_newHL AT %QL0.12 : LREAL;
      AI_Tstali_statora_kanal_2_newHW AT %QL0.18 : LREAL;
      AI_Tstali_statora_kanal_2_newLL AT %QL0.13 : LREAL;
      AI_Tstali_statora_kanal_2_status AT %QD0.15 : UDINT;
      AI_Tstali_statora_kanal_2_value AT %QL0.16 : LREAL;
      AI_Tstali_statora_kanal_3_HL AT %QL0.19 : LREAL;
      AI_Tstali_statora_kanal_3_HW AT %QL0.26 : LREAL;
      AI_Tstali_statora_kanal_3_LL AT %QL0.20 : LREAL;
      AI_Tstali_statora_kanal_3_command AT %QW0.23 : UINT;
      AI_Tstali_statora_kanal_3_newHL AT %QL0.21 : LREAL;
      AI_Tstali_statora_kanal_3_newHW AT %QL0.27 : LREAL;
      AI_Tstali_statora_kanal_3_newLL AT %QL0.22 : LREAL;
      AI_Tstali_statora_kanal_3_status AT %QD0.24 : UDINT;
      AI_Tstali_statora_kanal_3_value AT %QL0.25 : LREAL;
      AI_Ty_podshipnika_nagnet_EDT_7_1_HA AT %QL0.130 : LREAL;
      AI_Ty_podshipnika_nagnet_EDT_7_1_HL AT %QL0.121 : LREAL;
      AI_Ty_podshipnika_nagnet_EDT_7_1_HW AT %QL0.128 : LREAL;
      AI_Ty_podshipnika_nagnet_EDT_7_1_LL AT %QL0.122 : LREAL;
      AI_Ty_podshipnika_nagnet_EDT_7_1_command AT %QW0.125 : UINT;
      AI_Ty_podshipnika_nagnet_EDT_7_1_newHA AT %QL0.131 : LREAL;
      AI_Ty_podshipnika_nagnet_EDT_7_1_newHL AT %QL0.123 : LREAL;
      AI_Ty_podshipnika_nagnet_EDT_7_1_newHW AT %QL0.129 : LREAL;
      AI_Ty_podshipnika_nagnet_EDT_7_1_newLL AT %QL0.124 : LREAL;
      AI_Ty_podshipnika_nagnet_EDT_7_1_status AT %QD0.126 : UDINT;
      AI_Ty_podshipnika_nagnet_EDT_7_1_value AT %QL0.127 : LREAL;
      AI_Ty_podshipnika_nagnet_EDT_7_2_HA AT %QL0.141 : LREAL;
      AI_Ty_podshipnika_nagnet_EDT_7_2_HL AT %QL0.132 : LREAL;
      AI_Ty_podshipnika_nagnet_EDT_7_2_HW AT %QL0.139 : LREAL;
      AI_Ty_podshipnika_nagnet_EDT_7_2_LL AT %QL0.133 : LREAL;
      AI_Ty_podshipnika_nagnet_EDT_7_2_command AT %QW0.136 : UINT;
      AI_Ty_podshipnika_nagnet_EDT_7_2_newHA AT %QL0.142 : LREAL;
      AI_Ty_podshipnika_nagnet_EDT_7_2_newHL AT %QL0.134 : LREAL;
      AI_Ty_podshipnika_nagnet_EDT_7_2_newHW AT %QL0.140 : LREAL;
      AI_Ty_podshipnika_nagnet_EDT_7_2_newLL AT %QL0.135 : LREAL;
      AI_Ty_podshipnika_nagnet_EDT_7_2_status AT %QD0.137 : UDINT;
      AI_Ty_podshipnika_nagnet_EDT_7_2_value AT %QL0.138 : LREAL;
      AI_Ty_podshipnika_red_EDT_6_HA AT %QL0.119 : LREAL;
      AI_Ty_podshipnika_red_EDT_6_HL AT %QL0.110 : LREAL;
      AI_Ty_podshipnika_red_EDT_6_HW AT %QL0.117 : LREAL;
      AI_Ty_podshipnika_red_EDT_6_LL AT %QL0.111 : LREAL;
      AI_Ty_podshipnika_red_EDT_6_command AT %QW0.114 : UINT;
      AI_Ty_podshipnika_red_EDT_6_newHA AT %QL0.120 : LREAL;
      AI_Ty_podshipnika_red_EDT_6_newHL AT %QL0.112 : LREAL;
      AI_Ty_podshipnika_red_EDT_6_newHW AT %QL0.118 : LREAL;
      AI_Ty_podshipnika_red_EDT_6_newLL AT %QL0.113 : LREAL;
      AI_Ty_podshipnika_red_EDT_6_status AT %QD0.115 : UDINT;
      AI_Ty_podshipnika_red_EDT_6_value AT %QL0.116 : LREAL;
      AI_Vibro_skorost_OPED_T1_HA AT %QL0.967 : LREAL;
      AI_Vibro_skorost_OPED_T1_HL AT %QL0.958 : LREAL;
      AI_Vibro_skorost_OPED_T1_HW AT %QL0.965 : LREAL;
      AI_Vibro_skorost_OPED_T1_LL AT %QL0.959 : LREAL;
      AI_Vibro_skorost_OPED_T1_command AT %QW0.962 : UINT;
      AI_Vibro_skorost_OPED_T1_newHA AT %QL0.968 : LREAL;
      AI_Vibro_skorost_OPED_T1_newHL AT %QL0.960 : LREAL;
      AI_Vibro_skorost_OPED_T1_newHW AT %QL0.966 : LREAL;
      AI_Vibro_skorost_OPED_T1_newLL AT %QL0.961 : LREAL;
      AI_Vibro_skorost_OPED_T1_status AT %QD0.963 : UDINT;
      AI_Vibro_skorost_OPED_T1_value AT %QL0.964 : LREAL;
      AI_Vibro_skorost_OP_kolesa_RH_T4_HA AT %QL0.1000 : LREAL;
      AI_Vibro_skorost_OP_kolesa_RH_T4_HL AT %QL0.991 : LREAL;
      AI_Vibro_skorost_OP_kolesa_RH_T4_HW AT %QL0.998 : LREAL;
      AI_Vibro_skorost_OP_kolesa_RH_T4_LL AT %QL0.992 : LREAL;
      AI_Vibro_skorost_OP_kolesa_RH_T4_command AT %QW0.995 : UINT;
      AI_Vibro_skorost_OP_kolesa_RH_T4_newHA AT %QL0.1001 : LREAL;
      AI_Vibro_skorost_OP_kolesa_RH_T4_newHL AT %QL0.993 : LREAL;
      AI_Vibro_skorost_OP_kolesa_RH_T4_newHW AT %QL0.999 : LREAL;
      AI_Vibro_skorost_OP_kolesa_RH_T4_newLL AT %QL0.994 : LREAL;
      AI_Vibro_skorost_OP_kolesa_RH_T4_status AT %QD0.996 : UDINT;
      AI_Vibro_skorost_OP_kolesa_RH_T4_value AT %QL0.997 : LREAL;
      AI_Vibro_skorost_OP_shesterni_RED_T5_HA AT %QL0.1011 : LREAL;
      AI_Vibro_skorost_OP_shesterni_RED_T5_HL AT %QL0.1002 : LREAL;
      AI_Vibro_skorost_OP_shesterni_RED_T5_HW AT %QL0.1009 : LREAL;
      AI_Vibro_skorost_OP_shesterni_RED_T5_LL AT %QL0.1003 : LREAL;
      AI_Vibro_skorost_OP_shesterni_RED_T5_command AT %QW0.1006 : UINT;
      AI_Vibro_skorost_OP_shesterni_RED_T5_newHA AT %QL0.1012 : LREAL;
      AI_Vibro_skorost_OP_shesterni_RED_T5_newHL AT %QL0.1004 : LREAL;
      AI_Vibro_skorost_OP_shesterni_RED_T5_newHW AT %QL0.1010 : LREAL;
      AI_Vibro_skorost_OP_shesterni_RED_T5_newLL AT %QL0.1005 : LREAL;
      AI_Vibro_skorost_OP_shesterni_RED_T5_status AT %QD0.1007 : UDINT;
      AI_Vibro_skorost_OP_shesterni_RED_T5_value AT %QL0.1008 : LREAL;
      AI_Vibro_skorost_OP_shesterni_RED_T6_HA AT %QL0.1022 : LREAL;
      AI_Vibro_skorost_OP_shesterni_RED_T6_HL AT %QL0.1013 : LREAL;
      AI_Vibro_skorost_OP_shesterni_RED_T6_HW AT %QL0.1020 : LREAL;
      AI_Vibro_skorost_OP_shesterni_RED_T6_LL AT %QL0.1014 : LREAL;
      AI_Vibro_skorost_OP_shesterni_RED_T6_command AT %QW0.1017 : UINT;
      AI_Vibro_skorost_OP_shesterni_RED_T6_newHA AT %QL0.1023 : LREAL;
      AI_Vibro_skorost_OP_shesterni_RED_T6_newHL AT %QL0.1015 : LREAL;
      AI_Vibro_skorost_OP_shesterni_RED_T6_newHW AT %QL0.1021 : LREAL;
      AI_Vibro_skorost_OP_shesterni_RED_T6_newLL AT %QL0.1016 : LREAL;
      AI_Vibro_skorost_OP_shesterni_RED_T6_status AT %QD0.1018 : UDINT;
      AI_Vibro_skorost_OP_shesterni_RED_T6_value AT %QL0.1019 : LREAL;
      AI_Vibro_skorost_OYPED_T2_HA AT %QL0.978 : LREAL;
      AI_Vibro_skorost_OYPED_T2_HL AT %QL0.969 : LREAL;
      AI_Vibro_skorost_OYPED_T2_HW AT %QL0.976 : LREAL;
      AI_Vibro_skorost_OYPED_T2_LL AT %QL0.970 : LREAL;
      AI_Vibro_skorost_OYPED_T2_command AT %QW0.973 : UINT;
      AI_Vibro_skorost_OYPED_T2_newHA AT %QL0.979 : LREAL;
      AI_Vibro_skorost_OYPED_T2_newHL AT %QL0.971 : LREAL;
      AI_Vibro_skorost_OYPED_T2_newHW AT %QL0.977 : LREAL;
      AI_Vibro_skorost_OYPED_T2_newLL AT %QL0.972 : LREAL;
      AI_Vibro_skorost_OYPED_T2_status AT %QD0.974 : UDINT;
      AI_Vibro_skorost_OYPED_T2_value AT %QL0.975 : LREAL;
      AI_Vibro_skorost_OYP_kolesa_ED_T3_HA AT %QL0.989 : LREAL;
      AI_Vibro_skorost_OYP_kolesa_ED_T3_HL AT %QL0.980 : LREAL;
      AI_Vibro_skorost_OYP_kolesa_ED_T3_HW AT %QL0.987 : LREAL;
      AI_Vibro_skorost_OYP_kolesa_ED_T3_LL AT %QL0.981 : LREAL;
      AI_Vibro_skorost_OYP_kolesa_ED_T3_command AT %QW0.984 : UINT;
      AI_Vibro_skorost_OYP_kolesa_ED_T3_newHA AT %QL0.990 : LREAL;
      AI_Vibro_skorost_OYP_kolesa_ED_T3_newHL AT %QL0.982 : LREAL;
      AI_Vibro_skorost_OYP_kolesa_ED_T3_newHW AT %QL0.988 : LREAL;
      AI_Vibro_skorost_OYP_kolesa_ED_T3_newLL AT %QL0.983 : LREAL;
      AI_Vibro_skorost_OYP_kolesa_ED_T3_status AT %QD0.985 : UDINT;
      AI_Vibro_skorost_OYP_kolesa_ED_T3_value AT %QL0.986 : LREAL;
      AI_Yroven_masla_MB_HL AT %QL0.875 : LREAL;
      AI_Yroven_masla_MB_LL AT %QL0.876 : LREAL;
      AI_Yroven_masla_MB_LW AT %QL0.925 : LREAL;
      AI_Yroven_masla_MB_command AT %QW0.922 : UINT;
      AI_Yroven_masla_MB_newHL AT %QL0.877 : LREAL;
      AI_Yroven_masla_MB_newLL AT %QL0.921 : LREAL;
      AI_Yroven_masla_MB_newLW AT %QL0.926 : LREAL;
      AI_Yroven_masla_MB_status AT %QD0.923 : UDINT;
      AI_Yroven_masla_MB_value AT %QL0.924 : LREAL;
      AI_dPgaza_na_konfuzore_HL AT %QL0.397 : LREAL;
      AI_dPgaza_na_konfuzore_LL AT %QL0.398 : LREAL;
      AI_dPgaza_na_konfuzore_LW AT %QL0.404 : LREAL;
      AI_dPgaza_na_konfuzore_command AT %QW0.401 : UINT;
      AI_dPgaza_na_konfuzore_newHL AT %QL0.399 : LREAL;
      AI_dPgaza_na_konfuzore_newLL AT %QL0.400 : LREAL;
      AI_dPgaza_na_konfuzore_newLW AT %QL0.405 : LREAL;
      AI_dPgaza_na_konfuzore_status AT %QD0.402 : UDINT;
      AI_dPgaza_na_konfuzore_value AT %QL0.403 : LREAL;
      AI_dPgaza_na_maslo_filtre_HL AT %QL0.388 : LREAL;
      AI_dPgaza_na_maslo_filtre_HW AT %QL0.395 : LREAL;
      AI_dPgaza_na_maslo_filtre_LL AT %QL0.389 : LREAL;
      AI_dPgaza_na_maslo_filtre_command AT %QW0.392 : UINT;
      AI_dPgaza_na_maslo_filtre_newHL AT %QL0.390 : LREAL;
      AI_dPgaza_na_maslo_filtre_newHW AT %QL0.396 : LREAL;
      AI_dPgaza_na_maslo_filtre_newLL AT %QL0.391 : LREAL;
      AI_dPgaza_na_maslo_filtre_status AT %QD0.393 : UDINT;
      AI_dPgaza_na_maslo_filtre_value AT %QL0.394 : LREAL;
      AI_dPmaslo_gaz_HL AT %QL0.406 : LREAL;
      AI_dPmaslo_gaz_LA AT %QL0.415 : LREAL;
      AI_dPmaslo_gaz_LL AT %QL0.407 : LREAL;
      AI_dPmaslo_gaz_LW AT %QL0.413 : LREAL;
      AI_dPmaslo_gaz_command AT %QW0.410 : UINT;
      AI_dPmaslo_gaz_newHL AT %QL0.408 : LREAL;
      AI_dPmaslo_gaz_newLA AT %QL0.416 : LREAL;
      AI_dPmaslo_gaz_newLL AT %QL0.409 : LREAL;
      AI_dPmaslo_gaz_newLW AT %QL0.414 : LREAL;
      AI_dPmaslo_gaz_status AT %QD0.411 : UDINT;
      AI_dPmaslo_gaz_value AT %QL0.412 : LREAL;
      A1_10_err_mode AT %QW0.825 : UINT;
      A1_11_err_mode AT %QW0.826 : UINT;
      A1_12_err_mode AT %QW0.827 : UINT;
      A1_13_err_mode AT %QW0.828 : UINT;
      A1_14_err_mode AT %QW0.829 : UINT;
      A1_15_err_mode AT %QW0.830 : UINT;
      A1_1_err_mode AT %QW0.816 : UINT;
      A1_2_err_mode AT %QW0.817 : UINT;
      A1_3_err_mode AT %QW0.818 : UINT;
      A1_4_err_mode AT %QW0.819 : UINT;
      A1_5_err_mode AT %QW0.820 : UINT;
      A1_6_err_mode AT %QW0.821 : UINT;
      A1_7_err_mode AT %QW0.822 : UINT;
      A1_8_err_mode AT %QW0.823 : UINT;
      A1_9_err_mode AT %QW0.824 : UINT;
      A2_10_err_mode AT %QW0.840 : UINT;
      A2_11_err_mode AT %QW0.841 : UINT;
      A2_12_err_mode AT %QW0.842 : UINT;
      A2_13_err_mode AT %QW0.843 : UINT;
      A2_14_err_mode AT %QW0.844 : UINT;
      A2_15_err_mode AT %QW0.845 : UINT;
      A2_1_err_mode AT %QW0.831 : UINT;
      A2_2_err_mode AT %QW0.832 : UINT;
      A2_3_err_mode AT %QW0.833 : UINT;
      A2_4_err_mode AT %QW0.834 : UINT;
      A2_5_err_mode AT %QW0.835 : UINT;
      A2_6_err_mode AT %QW0.836 : UINT;
      A2_7_err_mode AT %QW0.837 : UINT;
      A2_8_err_mode AT %QW0.838 : UINT;
      A2_9_err_mode AT %QW0.839 : UINT;
      AI_0_dblValue AT %QL0.736 : LREAL;
      AI_10_dblValue AT %QL0.746 : LREAL;
      AI_11_dblValue AT %QL0.747 : LREAL;
      AI_12_dblValue AT %QL0.748 : LREAL;
      AI_13_dblValue AT %QL0.749 : LREAL;
      AI_14_dblValue AT %QL0.750 : LREAL;
      AI_15_dblValue AT %QL0.751 : LREAL;
      AI_16_dblValue AT %QL0.752 : LREAL;
      AI_17_dblValue AT %QL0.753 : LREAL;
      AI_18_dblValue AT %QL0.754 : LREAL;
      AI_19_dblValue AT %QL0.755 : LREAL;
      AI_1_dblValue AT %QL0.737 : LREAL;
      AI_20_dblValue AT %QL0.756 : LREAL;
      AI_21_dblValue AT %QL0.757 : LREAL;
      AI_22_dblValue AT %QL0.758 : LREAL;
      AI_23_dblValue AT %QL0.759 : LREAL;
      AI_24_dblValue AT %QL0.760 : LREAL;
      AI_25_dblValue AT %QL0.761 : LREAL;
      AI_26_dblValue AT %QL0.762 : LREAL;
      AI_27_dblValue AT %QL0.763 : LREAL;
      AI_28_dblValue AT %QL0.764 : LREAL;
      AI_29_dblValue AT %QL0.765 : LREAL;
      AI_2_dblValue AT %QL0.738 : LREAL;
      AI_30_dblValue AT %QL0.766 : LREAL;
      AI_31_dblValue AT %QL0.767 : LREAL;
      AI_32_dblValue AT %QL0.768 : LREAL;
      AI_33_dblValue AT %QL0.769 : LREAL;
      AI_34_dblValue AT %QL0.770 : LREAL;
      AI_35_dblValue AT %QL0.771 : LREAL;
      AI_36_dblValue AT %QL0.772 : LREAL;
      AI_37_dblValue AT %QL0.773 : LREAL;
      AI_38_dblValue AT %QL0.774 : LREAL;
      AI_39_dblValue AT %QL0.775 : LREAL;
      AI_3_dblValue AT %QL0.739 : LREAL;
      AI_40_dblValue AT %QL0.776 : LREAL;
      AI_41_dblValue AT %QL0.777 : LREAL;
      AI_42_dblValue AT %QL0.778 : LREAL;
      AI_43_dblValue AT %QL0.779 : LREAL;
      AI_44_dblValue AT %QL0.780 : LREAL;
      AI_45_dblValue AT %QL0.781 : LREAL;
      AI_46_dblValue AT %QL0.782 : LREAL;
      AI_47_dblValue AT %QL0.783 : LREAL;
      AI_48_dblValue AT %QL0.784 : LREAL;
      AI_49_dblValue AT %QL0.785 : LREAL;
      AI_4_dblValue AT %QL0.740 : LREAL;
      AI_50_dblValue AT %QL0.786 : LREAL;
      AI_51_dblValue AT %QL0.787 : LREAL;
      AI_52_dblValue AT %QL0.788 : LREAL;
      AI_53_dblValue AT %QL0.789 : LREAL;
      AI_54_dblValue AT %QL0.790 : LREAL;
      AI_55_dblValue AT %QL0.791 : LREAL;
      AI_56_dblValue AT %QL0.792 : LREAL;
      AI_57_dblValue AT %QL0.793 : LREAL;
      AI_58_dblValue AT %QL0.794 : LREAL;
      AI_59_dblValue AT %QL0.795 : LREAL;
      AI_5_dblValue AT %QL0.741 : LREAL;
      AI_60_dblValue AT %QL0.796 : LREAL;
      AI_61_dblValue AT %QL0.797 : LREAL;
      AI_62_dblValue AT %QL0.798 : LREAL;
      AI_63_dblValue AT %QL0.799 : LREAL;
      AI_64_dblValue AT %QL0.800 : LREAL;
      AI_65_dblValue AT %QL0.801 : LREAL;
      AI_66_dblValue AT %QL0.802 : LREAL;
      AI_67_dblValue AT %QL0.803 : LREAL;
      AI_68_dblValue AT %QL0.804 : LREAL;
      AI_69_dblValue AT %QL0.805 : LREAL;
      AI_6_dblValue AT %QL0.742 : LREAL;
      AI_70_dblValue AT %QL0.806 : LREAL;
      AI_71_dblValue AT %QL0.807 : LREAL;
      AI_72_dblValue AT %QL0.808 : LREAL;
      AI_73_dblValue AT %QL0.809 : LREAL;
      AI_74_dblValue AT %QL0.810 : LREAL;
      AI_75_dblValue AT %QL0.811 : LREAL;
      AI_76_dblValue AT %QL0.812 : LREAL;
      AI_77_dblValue AT %QL0.813 : LREAL;
      AI_78_dblValue AT %QL0.814 : LREAL;
      AI_79_dblValue AT %QL0.815 : LREAL;
      AI_7_dblValue AT %QL0.743 : LREAL;
      AI_8_dblValue AT %QL0.744 : LREAL;
      AI_9_dblValue AT %QL0.745 : LREAL;
      BS_Core1 AT %QD0.603 : REAL;
      BS_Core2 AT %QD0.675 : REAL;
      BS_Core3 AT %QD0.683 : REAL;
      BS_Core4 AT %QD0.709 : REAL;
      BS_FreeMemory AT %QD0.730 : REAL;
      BS_Temp1 AT %QD0.734 : REAL;
      BS_Temp2 AT %QD0.735 : REAL;
      DI_0_1_wValue AT %QD0.852 : UDINT;
      DI_10_11_wValue AT %QD0.857 : UDINT;
      DI_12_13_wValue AT %QD0.858 : UDINT;
      DI_14_15_wValue AT %QD0.859 : UDINT;
      DI_16_17_wValue AT %QD0.860 : UDINT;
      DI_18_19_wValue AT %QD0.861 : UDINT;
      DI_20_21_wValue AT %QD0.862 : UDINT;
      DI_2_3_wValue AT %QD0.853 : UDINT;
      DI_4_5_wValue AT %QD0.854 : UDINT;
      DI_6_7_wValue AT %QD0.855 : UDINT;
      DI_8_9_wValue AT %QD0.856 : UDINT;
      DO_0_wValue AT %QW0.846 : UINT;
      DO_1_wValue AT %QW0.847 : UINT;
      DO_2_wValue AT %QW0.848 : UINT;
      DO_3_wValue AT %QW0.849 : UINT;
      DO_4_wValue AT %QW0.850 : UINT;
      DO_5_wValue AT %QW0.851 : UINT;
      IM_CMN_inCommand_ARM AT %QW0.459 : UINT;
      IM_CMN_status AT %QD0.460 : UDINT;
      IM_KaloriferAVOM_inCommand_ARM AT %QW0.457 : UINT;
      IM_KaloriferAVOM_status AT %QD0.458 : UDINT;
      IM_Kran1_inCommand_ARM AT %QW0.427 : UINT;
      IM_Kran1_status AT %QD0.428 : UDINT;
      IM_Kran2_inCommand_ARM AT %QW0.429 : UINT;
      IM_Kran2_status AT %QD0.430 : UDINT;
      IM_Kran3_inCommand_ARM AT %QW0.431 : UINT;
      IM_Kran3_status AT %QD0.432 : UDINT;
      IM_Kran3b_inCommand_ARM AT %QW0.433 : UINT;
      IM_Kran3b_status AT %QD0.434 : UDINT;
      IM_Kran4_inCommand_ARM AT %QW0.435 : UINT;
      IM_Kran4_status AT %QD0.436 : UDINT;
      IM_Kran5_inCommand_ARM AT %QW0.437 : UINT;
      IM_Kran5_status AT %QD0.438 : UDINT;
      IM_Kran6_inCommand_ARM AT %QW0.439 : UINT;
      IM_Kran6_status AT %QD0.440 : UDINT;
      IM_SingleSignals_AO_GPA_ot_PRU_status AT %QD0.509 : UDINT;
      IM_SingleSignals_AO_GPA_ot_SHU_status AT %QD0.500 : UDINT;
      IM_SingleSignals_AO_KC_ot_SHKS_status AT %QD0.499 : UDINT;
      IM_SingleSignals_Assinhronnii_hod_peregruzka_status AT %QD0.474 : UDINT;
      IM_SingleSignals_Avariinoe_otkluch_vikluchatelya_status AT %QD0.473 : UDINT;
      IM_SingleSignals_BEAO_srabotal_status AT %QD0.501 : UDINT;
      IM_SingleSignals_Chastotny_pusk_status AT %QD0.502 : UDINT;
      IM_SingleSignals_Dver_SHU_pered_otkrita_status AT %QD0.667 : UDINT;
      IM_SingleSignals_Dver_SHU_zad_otkrita_status AT %QD0.668 : UDINT;
      IM_SingleSignals_EO_EGPA_ot_PRY_status AT %QD0.670 : UDINT;
      IM_SingleSignals_EO_GPA_ot_knopki_SHU_status AT %QD0.669 : UDINT;
      IM_SingleSignals_NKU1_GPA_on_status AT %QD0.497 : UDINT;
      IM_SingleSignals_NKU2_GPA_on_status AT %QD0.498 : UDINT;
      IM_SingleSignals_NO_GPA_ot_SHU_status AT %QD0.508 : UDINT;
      IM_SingleSignals_NS_G10_G11_status AT %QD0.494 : UDINT;
      IM_SingleSignals_NS_G13_G14_status AT %QD0.495 : UDINT;
      IM_SingleSignals_NS_G15_G16_status AT %QD0.489 : UDINT;
      IM_SingleSignals_NS_G17_status AT %QD0.490 : UDINT;
      IM_SingleSignals_NS_G18_G19_status AT %QD0.493 : UDINT;
      IM_SingleSignals_NS_G1_G2_status AT %QD0.487 : UDINT;
      IM_SingleSignals_NS_G3_G4_status AT %QD0.488 : UDINT;
      IM_SingleSignals_NS_G5_G6_status AT %QD0.491 : UDINT;
      IM_SingleSignals_NS_G7_G8_status AT %QD0.492 : UDINT;
      IM_SingleSignals_Nalichie_220BEAO_status AT %QD0.519 : UDINT;
      IM_SingleSignals_Nalichie_BP11_status AT %QD0.665 : UDINT;
      IM_SingleSignals_Nalichie_BP12_status AT %QD0.666 : UDINT;
      IM_SingleSignals_Nalichie_BP1_status AT %QD0.510 : UDINT;
      IM_SingleSignals_Nalichie_BP2_status AT %QD0.511 : UDINT;
      IM_SingleSignals_Nalichie_BP3_status AT %QD0.512 : UDINT;
      IM_SingleSignals_Nalichie_BP4_status AT %QD0.513 : UDINT;
      IM_SingleSignals_Nalichie_BP5_status AT %QD0.514 : UDINT;
      IM_SingleSignals_Nalichie_BP6_status AT %QD0.515 : UDINT;
      IM_SingleSignals_Nalichie_BP7_BP8_status AT %QD0.516 : UDINT;
      IM_SingleSignals_Nalichie_BP9_BP10_status AT %QD0.517 : UDINT;
      IM_SingleSignals_Nalichie_cepei_upravlen_mv_status AT %QD0.518 : UDINT;
      IM_SingleSignals_Nalichie_per_220_na_vhode_status AT %QD0.663 : UDINT;
      IM_SingleSignals_Nalichie_post_220_na_vhode_status AT %QD0.664 : UDINT;
      IM_SingleSignals_Neuspesh_chastotny_pusk_status AT %QD0.503 : UDINT;
      IM_SingleSignals_Osnovnoy_regul_off_status AT %QD0.505 : UDINT;
      IM_SingleSignals_Potok_ms_posle_AVOM_status AT %QD0.672 : UDINT;
      IM_SingleSignals_QF10_QF11_on_status AT %QD0.483 : UDINT;
      IM_SingleSignals_QF12_QF13_on_status AT %QD0.484 : UDINT;
      IM_SingleSignals_QF14_QF15_on_status AT %QD0.485 : UDINT;
      IM_SingleSignals_QF1_on_status AT %QD0.477 : UDINT;
      IM_SingleSignals_QF22_on_status AT %QD0.486 : UDINT;
      IM_SingleSignals_QF23_on_status AT %QD0.479 : UDINT;
      IM_SingleSignals_QF2_on_status AT %QD0.478 : UDINT;
      IM_SingleSignals_QF4_QF5_on_status AT %QD0.480 : UDINT;
      IM_SingleSignals_QF6_QF7_on_status AT %QD0.481 : UDINT;
      IM_SingleSignals_QF8_QF9_on_status AT %QD0.482 : UDINT;
      IM_SingleSignals_Razreshenie_zagruzki_dvig_status AT %QD0.467 : UDINT;
      IM_SingleSignals_Reactorny_pusk_status AT %QD0.507 : UDINT;
      IM_SingleSignals_Rezhim_ruchnogo_regulirovaniya_status AT %QD0.504 : UDINT;
      IM_SingleSignals_SHAVR1_v_rabote_status AT %QD0.471 : UDINT;
      IM_SingleSignals_SHAVR2_v_rabote_status AT %QD0.472 : UDINT;
      IM_SingleSignals_SHP_v_GPA_vkluch_status AT %QD0.476 : UDINT;
      IM_SingleSignals_SHU_v_GPA_vkluch_status AT %QD0.475 : UDINT;
      IM_SingleSignals_Synchroniz_rezhima_K1_status AT %QD0.671 : UDINT;
      IM_SingleSignals_Uroven_masla_akkum_status AT %QD0.496 : UDINT;
      IM_SingleSignals_Voltage_sekcii_norm_status AT %QD0.506 : UDINT;
      IM_SingleSignals_Vozbud_gotovnost_status AT %QD0.468 : UDINT;
      IM_SingleSignals_Vozbud_neispr_tsepey_upr_AVR_pit_status AT %QD0.469 : UDINT;
      IM_SingleSignals_Vozbud_neispravnost_status AT %QD0.470 : UDINT;
      IM_SingleSignals_dP_maslo_gaz_Less100_status AT %QD0.465 : UDINT;
      IM_SingleSignals_dp_kran1_Less100_status AT %QD0.466 : UDINT;
      IM_TEN_MB_inCommand_ARM AT %QW0.463 : UINT;
      IM_TEN_MB_status AT %QD0.464 : UDINT;
      IM_TEN_kollectora_inCommand_ARM AT %QW0.461 : UINT;
      IM_TEN_kollectora_status AT %QD0.462 : UDINT;
      IM_mv_inCommand_ARM AT %QW0.455 : UINT;
      IM_mv_status AT %QD0.456 : UDINT;
      IM_nu1_inCommand_ARM AT %QW0.441 : UINT;
      IM_nu1_status AT %QD0.442 : UDINT;
      IM_nu2_inCommand_ARM AT %QW0.443 : UINT;
      IM_nu2_status AT %QD0.444 : UDINT;
      IM_pns_inCommand_ARM AT %QW0.445 : UINT;
      IM_pns_status AT %QD0.446 : UDINT;
      IM_v1_Avom_inCommand_ARM AT %QW0.447 : UINT;
      IM_v1_Avom_status AT %QD0.448 : UDINT;
      IM_v2_Avom_inCommand_ARM AT %QW0.449 : UINT;
      IM_v2_Avom_status AT %QD0.450 : UDINT;
      IM_v3_Avom_inCommand_ARM AT %QW0.451 : UINT;
      IM_v3_Avom_status AT %QD0.452 : UDINT;
      IM_v4_Avom_inCommand_ARM AT %QW0.453 : UINT;
      IM_v4_Avom_status AT %QD0.454 : UDINT;
      algoritms_AntiPompag AT %QW0.895 : UINT;
      algoritms_Apusk AT %QW0.905 : UINT;
      algoritms_AutoAvom AT %QW0.893 : UINT;
      algoritms_AutoPns AT %QW0.892 : UINT;
      algoritms_AutoTen AT %QW0.894 : UINT;
      algoritms_LineToRing AT %QW0.903 : UINT;
      algoritms_Prov_PMS_ALG AT %QW0.917 : UINT;
      algoritms_Prov_opressovka_ALG AT %QW0.918 : UINT;
      algoritms_Pusk_F_faza1 AT %QW0.914 : UINT;
      algoritms_Pusk_F_faza2 AT %QW0.915 : UINT;
      algoritms_Pusk_SEC_faza_chastotny AT %QW0.919 : UINT;
      algoritms_Pusk_SEC_faza_reactor AT %QW0.920 : UINT;
      algoritms_Pusk_TH_faza AT %QW0.916 : UINT;
      algoritms_Remont AT %QW0.898 : UINT;
      algoritms_RingToLine AT %QW0.904 : UINT;
      algoritms_SemiAutoPusk AT %QW0.906 : UINT;
      algoritms_TestProtection AT %QW0.897 : UINT;
      algoritms_ao AT %QW0.909 : UINT;
      algoritms_engineRun AT %QW0.901 : UINT;
      algoritms_filling AT %QW0.902 : UINT;
      algoritms_no AT %QW0.907 : UINT;
      algoritms_ppu AT %QW0.899 : UINT;
      algoritms_puskK AT %QW0.913 : UINT;
      algoritms_puskOilSystem AT %QW0.900 : UINT;
      algoritms_puskV AT %QW0.912 : UINT;
      algoritms_testIm AT %QW0.896 : UINT;
      algoritms_testPms AT %QW0.910 : UINT;
      algoritms_testdPmg AT %QW0.911 : UINT;
      algoritms_vibegPNS AT %QW0.908 : UINT;
      algManager_Mode AT %QW0.610 : UINT;
      algoritms_AntiPompag_command AT %QW0.631 : UINT;
      algoritms_Apusk_Error AT %QD0.564 : UDINT;
      algoritms_Apusk_Start AT %QD0.565 : UDINT;
      algoritms_Apusk_Top AT %QD0.566 : UDINT;
      algoritms_Apusk_command AT %QW0.641 : UINT;
      algoritms_Apusk_status AT %QD0.567 : UDINT;
      algoritms_AutoAvom_Error AT %ID0.661 : UDINT;
      algoritms_AutoAvom_Start AT %ID0.660 : UDINT;
      algoritms_AutoAvom_Top AT %ID0.662 : UDINT;
      algoritms_AutoAvom_command AT %QW0.629 : UINT;
      algoritms_AutoAvom_status AT %QD0.520 : UDINT;
      algoritms_AutoPns_OffTimer AT %QW0.611 : UINT;
      algoritms_AutoPns_OnTimer AT %QW0.612 : UINT;
      algoritms_AutoPns_command AT %QW0.628 : UINT;
      algoritms_AutoPns_status AT %QD0.521 : UDINT;
      algoritms_AutoTen_command AT %QW0.630 : UINT;
      algoritms_AutoTen_status AT %QD0.522 : UDINT;
      algoritms_LineToRing_command AT %QW0.639 : UINT;
      algoritms_Prov_PMS_ALG_Error AT %QD0.539 : UDINT;
      algoritms_Prov_PMS_ALG_Start AT %QD0.540 : UDINT;
      algoritms_Prov_PMS_ALG_Top AT %QD0.538 : UDINT;
      algoritms_Prov_PMS_ALG_command AT %QW0.653 : UINT;
      algoritms_Prov_PMS_ALG_status AT %QD0.541 : UDINT;
      algoritms_Prov_opressovka_ALG_Error AT %QD0.535 : UDINT;
      algoritms_Prov_opressovka_ALG_Start AT %QD0.536 : UDINT;
      algoritms_Prov_opressovka_ALG_Top AT %QD0.534 : UDINT;
      algoritms_Prov_opressovka_ALG_command AT %QW0.654 : UINT;
      algoritms_Prov_opressovka_ALG_status AT %QD0.537 : UDINT;
      algoritms_Pusk_F_faza1_Error AT %QD0.551 : UDINT;
      algoritms_Pusk_F_faza1_Start AT %QD0.552 : UDINT;
      algoritms_Pusk_F_faza1_Top AT %QD0.550 : UDINT;
      algoritms_Pusk_F_faza1_command AT %QW0.650 : UINT;
      algoritms_Pusk_F_faza1_status AT %QD0.553 : UDINT;
      algoritms_Pusk_F_faza2_Error AT %QD0.547 : UDINT;
      algoritms_Pusk_F_faza2_Start AT %QD0.548 : UDINT;
      algoritms_Pusk_F_faza2_Top AT %QD0.546 : UDINT;
      algoritms_Pusk_F_faza2_command AT %QW0.651 : UINT;
      algoritms_Pusk_F_faza2_status AT %QD0.549 : UDINT;
      algoritms_Pusk_SEC_faza_chastotny_Error AT %QD0.531 : UDINT;
      algoritms_Pusk_SEC_faza_chastotny_Start AT %QD0.532 : UDINT;
      algoritms_Pusk_SEC_faza_chastotny_Top AT %QD0.530 : UDINT;
      algoritms_Pusk_SEC_faza_chastotny_command AT %QW0.655 : UINT;
      algoritms_Pusk_SEC_faza_chastotny_status AT %QD0.533 : UDINT;
      algoritms_Pusk_SEC_faza_reactor_Error AT %QD0.527 : UDINT;
      algoritms_Pusk_SEC_faza_reactor_Start AT %QD0.528 : UDINT;
      algoritms_Pusk_SEC_faza_reactor_Top AT %QD0.526 : UDINT;
      algoritms_Pusk_SEC_faza_reactor_command AT %QW0.656 : UINT;
      algoritms_Pusk_SEC_faza_reactor_status AT %QD0.529 : UDINT;
      algoritms_Pusk_TH_faza_Error AT %QD0.543 : UDINT;
      algoritms_Pusk_TH_faza_Start AT %QD0.544 : UDINT;
      algoritms_Pusk_TH_faza_Top AT %QD0.542 : UDINT;
      algoritms_Pusk_TH_faza_command AT %QW0.652 : UINT;
      algoritms_Pusk_TH_faza_status AT %QD0.545 : UDINT;
      algoritms_Remont_command AT %QW0.634 : UINT;
      algoritms_Remont_status AT %QD0.523 : UDINT;
      algoritms_RingToLine_Error AT %QD0.568 : UDINT;
      algoritms_RingToLine_Start AT %QD0.569 : UDINT;
      algoritms_RingToLine_Top AT %QD0.570 : UDINT;
      algoritms_RingToLine_command AT %QW0.640 : UINT;
      algoritms_RingToLine_status AT %QD0.571 : UDINT;
      algoritms_SemiAutoPusk_command AT %QW0.642 : UINT;
      algoritms_TestProtection_command AT %QW0.633 : UINT;
      algoritms_TestProtection_status AT %QD0.524 : UDINT;
      algoritms_ao_Error AT %QD0.572 : UDINT;
      algoritms_ao_Start AT %QD0.573 : UDINT;
      algoritms_ao_Top AT %QD0.574 : UDINT;
      algoritms_ao_command AT %QW0.645 : UINT;
      algoritms_ao_status AT %QD0.575 : UDINT;
      algoritms_ao_waitKran_timer AT %QW0.613 : UINT;
      algoritms_autoNu AT %QW0.891 : UINT;
      algoritms_autoNu_Error AT %ID0.658 : UDINT;
      algoritms_autoNu_NotHasRezervNU AT %QX0.626 : BOOL;
      algoritms_autoNu_Start AT %ID0.657 : UDINT;
      algoritms_autoNu_Top AT %ID0.659 : UDINT;
      algoritms_autoNu_command AT %QW0.627 : UINT;
      algoritms_autoNu_status AT %QD0.525 : UDINT;
      algoritms_engineRun_BreakPuskTimer_timer AT %QW0.614 : UINT;
      algoritms_engineRun_Error AT %QD0.576 : UDINT;
      algoritms_engineRun_Start AT %QD0.577 : UDINT;
      algoritms_engineRun_Top AT %QD0.578 : UDINT;
      algoritms_engineRun_command AT %QW0.637 : UINT;
      algoritms_engineRun_status AT %QD0.579 : UDINT;
      algoritms_filling_BreakPuskTimer_timer AT %QW0.615 : UINT;
      algoritms_filling_Error AT %QD0.580 : UDINT;
      algoritms_filling_Start AT %QD0.581 : UDINT;
      algoritms_filling_Top AT %QD0.582 : UDINT;
      algoritms_filling_command AT %QW0.638 : UINT;
      algoritms_filling_status AT %QD0.583 : UDINT;
      algoritms_filling_waitAfterKran4_timer AT %QW0.616 : UINT;
      algoritms_filling_waitAfterKran5_timer AT %QW0.617 : UINT;
      algoritms_no_Error AT %QD0.584 : UDINT;
      algoritms_no_Start AT %QD0.585 : UDINT;
      algoritms_no_Top AT %QD0.586 : UDINT;
      algoritms_no_command AT %QW0.643 : UINT;
      algoritms_no_status AT %QD0.587 : UDINT;
      algoritms_no_waitCloseKran_timer AT %QW0.618 : UINT;
      algoritms_ppu_Error AT %QD0.588 : UDINT;
      algoritms_ppu_Start AT %QD0.589 : UDINT;
      algoritms_ppu_Top AT %QD0.590 : UDINT;
      algoritms_ppu_command AT %QW0.635 : UINT;
      algoritms_ppu_status AT %QD0.591 : UDINT;
      algoritms_puskK_Error AT %QD0.592 : UDINT;
      algoritms_puskK_Start AT %QD0.593 : UDINT;
      algoritms_puskK_Top AT %QD0.594 : UDINT;
      algoritms_puskK_command AT %QW0.649 : UINT;
      algoritms_puskK_questionFilling_status AT %QD0.595 : UDINT;
      algoritms_puskK_questionUnload_status AT %QD0.596 : UDINT;
      algoritms_puskK_status AT %QD0.597 : UDINT;
      algoritms_puskK_wait720_timer AT %QW0.619 : UINT;
      algoritms_puskOilSystem_BreakPuskTimer_Poil_timer AT %QW0.620 : UINT;
      algoritms_puskOilSystem_BreakPuskTimer_dPmg_timer AT %QW0.621 : UINT;
      algoritms_puskOilSystem_Error AT %QD0.554 : UDINT;
      algoritms_puskOilSystem_Start AT %QD0.555 : UDINT;
      algoritms_puskOilSystem_Top AT %QD0.556 : UDINT;
      algoritms_puskOilSystem_command AT %QW0.636 : UINT;
      algoritms_puskOilSystem_status AT %QD0.557 : UDINT;
      algoritms_puskV_command AT %QW0.648 : UINT;
      algoritms_testIm_command AT %QW0.632 : UINT;
      algoritms_testIm_status AT %QD0.558 : UDINT;
      algoritms_testPms_BreakTest_timer AT %QW0.622 : UINT;
      algoritms_testPms_Error AT %QD0.598 : UDINT;
      algoritms_testPms_Start AT %QD0.599 : UDINT;
      algoritms_testPms_Top AT %QD0.600 : UDINT;
      algoritms_testPms_algContinue_status AT %QD0.601 : UDINT;
      algoritms_testPms_command AT %QW0.646 : UINT;
      algoritms_testPms_status AT %QD0.602 : UDINT;
      algoritms_testdPmg_BreakTest_timer AT %QW0.623 : UINT;
      algoritms_testdPmg_Error AT %QD0.604 : UDINT;
      algoritms_testdPmg_Start AT %QD0.605 : UDINT;
      algoritms_testdPmg_Top AT %QD0.606 : UDINT;
      algoritms_testdPmg_algContinue_status AT %QD0.607 : UDINT;
      algoritms_testdPmg_command AT %QW0.647 : UINT;
      algoritms_testdPmg_status AT %QD0.608 : UDINT;
      algoritms_vibegPNS_Error AT %QD0.559 : UDINT;
      algoritms_vibegPNS_Start AT %QD0.560 : UDINT;
      algoritms_vibegPNS_Top AT %QD0.561 : UDINT;
      algoritms_vibegPNS_algContinue_status AT %QD0.562 : UDINT;
      algoritms_vibegPNS_command AT %QW0.644 : UINT;
      algoritms_vibegPNS_status AT %QD0.563 : UDINT;
      algoritms_vibegPNS_waitVibeg_timer AT %QW0.609 : UINT;
      protectManager_protectionInRemont AT %QX0.624 : BOOL;
      protections_AOKC_SHKC_inCommand_ARM AT %QW0.879 : UINT;
      protections_AOKC_SHKC_status AT %QD0.880 : UDINT;
      protections_AO_PRU_inCommand_ARM AT %QW0.881 : UINT;
      protections_AO_PRU_status AT %QD0.882 : UDINT;
      protections_AO_ot_SHU_inCommand_ARM AT %QW0.883 : UINT;
      protections_AO_ot_SHU_status AT %QD0.884 : UDINT;
      protections_Fail_chastotnii_pusk_inCommand_ARM AT %QW0.731 : UINT;
      protections_Fail_chastotnii_pusk_status AT %QD0.732 : UDINT;
      protections_Kran1_sdvig_inCommand_ARM AT %QW0.887 : UINT;
      protections_Kran1_sdvig_status AT %QD0.888 : UDINT;
      protections_Kran2_sdvig_inCommand_ARM AT %QW0.889 : UINT;
      protections_Kran2_sdvig_status AT %QD0.890 : UDINT;
      protections_Off_avar_vikluchatel_inCommand_ARM AT %QW0.733 : UINT;
      protections_Off_avar_vikluchatel_status AT %QD0.878 : UDINT;
      protections_Os_sdvig_nagnetatelja_minus_inCommand_ARM AT %QW0.699 : UINT;
      protections_Os_sdvig_nagnetatelja_minus_status AT %QD0.700 : UDINT;
      protections_Os_sdvig_nagnetatelja_plus_inCommand_ARM AT %QW0.697 : UINT;
      protections_Os_sdvig_nagnetatelja_plus_status AT %QD0.698 : UDINT;
      protections_Pgaza_na_vhode_nagnetatelia_GPA_STOP_inCommand_ARM AT %QW0.703 : UINT;
      protections_Pgaza_na_vhode_nagnetatelia_GPA_STOP_status AT %QD0.704 : UDINT;
      protections_Pgaza_na_vyhode_nagnetatelia_GPA_STOP_inCommand_ARM AT %QW0.701 : UINT;
      protections_Pgaza_na_vyhode_nagnetatelia_GPA_STOP_status AT %QD0.702 : UDINT;
      protections_Pgaza_na_vyhode_nagnetatelia_inCommand_ARM AT %QW0.705 : UINT;
      protections_Pgaza_na_vyhode_nagnetatelia_status AT %QD0.706 : UDINT;
      protections_Pmaslo_sm_nizkoe_inCommand_ARM AT %QW0.710 : UINT;
      protections_Pmaslo_sm_nizkoe_status AT %QD0.711 : UDINT;
      protections_Pmaslo_sm_vysokoe_inCommand_ARM AT %QW0.712 : UINT;
      protections_Pmaslo_sm_vysokoe_status AT %QD0.713 : UDINT;
      protections_Reg_vozb_off_inCommand_ARM AT %QW0.728 : UINT;
      protections_Reg_vozb_off_status AT %QD0.729 : UDINT;
      protections_Tgaza_na_vyhode_H_inCommand_ARM AT %QW0.695 : UINT;
      protections_Tgaza_na_vyhode_H_status AT %QD0.696 : UDINT;
      protections_To_podshipnika_N_EDT_7_inCommand_ARM AT %QW0.687 : UINT;
      protections_To_podshipnika_N_EDT_7_status AT %QD0.688 : UDINT;
      protections_To_podshipnika_shest_red_EDT_5_inCommand_ARM AT %QW0.682 : UINT;
      protections_To_podshipnika_shest_red_EDT_5_status AT %QD0.684 : UDINT;
      protections_To_podshipnika_shest_red_EDT_6_inCommand_ARM AT %QW0.685 : UINT;
      protections_To_podshipnika_shest_red_EDT_6_status AT %QD0.686 : UDINT;
      protections_To_podshipnika_svob_konca_EDT_8_inCommand_ARM AT %QW0.689 : UINT;
      protections_To_podshipnika_svob_konca_EDT_8_status AT %QD0.690 : UDINT;
      protections_Topornogo_podshipnika_EDT_1_inCommand_ARM AT %QW0.673 : UINT;
      protections_Topornogo_podshipnika_EDT_1_status AT %QD0.674 : UDINT;
      protections_Toy_podshipnika_EDT_2_inCommand_ARM AT %QW0.676 : UINT;
      protections_Toy_podshipnika_EDT_2_status AT %QD0.677 : UDINT;
      protections_Toy_podshipnika_kol_EDT_3_inCommand_ARM AT %QW0.678 : UINT;
      protections_Toy_podshipnika_kol_EDT_3_status AT %QD0.679 : UDINT;
      protections_Toy_podshipnika_kol_EDT_4_inCommand_ARM AT %QW0.680 : UINT;
      protections_Toy_podshipnika_kol_EDT_4_status AT %QD0.681 : UDINT;
      protections_Ty_podshipnika_rab_kol_EDT_9_inCommand_ARM AT %QW0.691 : UINT;
      protections_Ty_podshipnika_rab_kol_EDT_9_status AT %QD0.692 : UDINT;
      protections_Typornogo_podshipnika_nerab_kolodok_HT_10_inCommand_ARM AT %QW0.693 : UINT;
      protections_Typornogo_podshipnika_nerab_kolodok_HT_10_status AT %QD0.694 : UDINT;
      protections_Vibro_skorost_OPED_T1_inCommand_ARM AT %QW0.714 : UINT;
      protections_Vibro_skorost_OPED_T1_status AT %QD0.715 : UDINT;
      protections_Vibro_skorost_OPED_T2_inCommand_ARM AT %QW0.716 : UINT;
      protections_Vibro_skorost_OPED_T2_status AT %QD0.717 : UDINT;
      protections_Vibro_skorost_OP_kolesa_RH_T4_inCommand_ARM AT %QW0.720 : UINT;
      protections_Vibro_skorost_OP_kolesa_RH_T4_status AT %QD0.721 : UDINT;
      protections_Vibro_skorost_OP_shesterni_RED_T5_inCommand_ARM AT %QW0.722 : UINT;
      protections_Vibro_skorost_OP_shesterni_RED_T5_status AT %QD0.723 : UDINT;
      protections_Vibro_skorost_OP_shesterni_RED_T6_inCommand_ARM AT %QW0.724 : UINT;
      protections_Vibro_skorost_OP_shesterni_RED_T6_status AT %QD0.725 : UDINT;
      protections_Vibro_skorost_OYP_kolesa_ED_T3_inCommand_ARM AT %QW0.718 : UINT;
      protections_Vibro_skorost_OYP_kolesa_ED_T3_status AT %QD0.719 : UDINT;
      protections_dPmaslo_gaz_inCommand_ARM AT %QW0.707 : UINT;
      protections_dPmaslo_gaz_less100_inCommand_ARM AT %QW0.726 : UINT;
      protections_dPmaslo_gaz_less100_status AT %QD0.727 : UDINT;
      protections_dPmaslo_gaz_status AT %QD0.708 : UDINT;
      protections_mvOff_inCommand_ARM AT %QW0.885 : UINT;
      protections_mvOff_status AT %QD0.886 : UDINT;
    END_VAR
    TASK task0(INTERVAL := T#20ms,PRIORITY := 0);
    PROGRAM instance0 WITH task0 : program0;
  END_RESOURCE
END_CONFIGURATION
